// TIA Portal project "智能仓库" (V16)

(* hardware
DEVICE "S7-1200 station_1"  S7-1200 Station
   slot 0: "Rack_0"  S7-1200 Rack  Rack  V1.0
   slot 1: "PLC_1"  CPU 1214C DC/DC/Rly  6ES7 214-1HG40-0XB0  V4.4
DEVICE "HMI_2"  TP700 Comfort
   slot 0: "HMI_2"  TP700 Comfort  6AV2 124-0GC01-0AX0  16.0.0.0
   slot 1: "HMI_RT_2"  TP700 Comfort  6AV2 124-0GC01-0AX0  16.0.0.0
   slot 5: "HMI_2.IE_CP_1"  PROFINET Interface  16.0.0.0
      slot 1: "PROFINET Interface_1"  PROFINET Interface
         slot 1: "Port_1"  Port
         slot 2: "Port_2"  Port
   slot 7: "HMI_2.MPI/DP_CP_1"  MPI/DP Interface  16.0.0.0
*)

// ===== PLC "PLC_1"  CPU 1214C DC/DC/Rly =====

VAR_GLOBAL   // PLC tag table "默认变量表"
   "System_Byte" AT %MB1 : Byte;
   "FirstScan" AT %M1.0 : Bool;
   "DiagStatusUpdate" AT %M1.1 : Bool;
   "AlwaysTRUE" AT %M1.2 : Bool;
   "AlwaysFALSE" AT %M1.3 : Bool;
   "System_Byte(1)" AT %MB1 : Byte;
   "Clock_Byte" AT %MB0 : Byte;
   "Clock_10Hz" AT %M0.0 : Bool;
   "Clock_5Hz" AT %M0.1 : Bool;
   "Clock_2.5Hz" AT %M0.2 : Bool;
   "Clock_2Hz" AT %M0.3 : Bool;
   "Clock_1.25Hz" AT %M0.4 : Bool;
   "Clock_1Hz" AT %M0.5 : Bool;
   "Clock_0.625Hz" AT %M0.6 : Bool;
   "Clock_0.5Hz" AT %M0.7 : Bool;
   "入库手/自动开关" AT %M10.0 : Bool;
   "自动入库读取当前数组的数据" AT %MB30 : Byte;
   "手动入库读取当前数组的数据" AT %MB34 : Byte;
   "动画列表" AT %MW100 : Int;
   "自动运行指示灯" AT %M10.1 : Bool;
   "手动运行指示灯" AT %M10.2 : Bool;
   "手动出库读取当前数组的数据" AT %MB38 : Byte;
   "自动出库读取当前数组的数据" AT %MB42 : Byte;
   "出库/入库切换开关" AT %M10.3 : Bool;
   "入库指示灯" AT %M10.4 : Bool;
   "出库指示灯" AT %M10.5 : Bool;
   "自动/手动出库开关" AT %M10.6 : Bool;
   "手动出库指示灯" AT %M10.7 : Bool;
   "自动出库指示灯" AT %M11.0 : Bool;
   "启动入库" AT %M100.0 : Bool;
   "启动出库" AT %M100.1 : Bool;
END_VAR

VAR_GLOBAL   // PLC tag table "factory  io"
   "伸出收料到位" AT %I2.0 : Bool;
   "叉车在中间" AT %I2.1 : Bool;
   "伸出放料到位" AT %I2.2 : Bool;
   "物料到位检测信号" AT %I2.3 : Bool;
   "检测物料开关" AT %I2.4 : Bool;
   "MovingX" AT %I2.5 : Bool;
   "Moving Z" AT %I2.6 : Bool;
   "启动" AT %I2.7 : Bool;
   "停止" AT %I3.0 : Bool;
   "出料检测传感器" AT %I3.1 : Bool;
   "显示屏传感器" AT %I3.2 : Bool;
   "复位" AT %I3.3 : Bool;
   "急停" AT %I3.4 : Bool;
   "手动模式" AT %I3.5 : Bool;
   "自动模式" AT %I3.6 : Bool;
   "FACTORY I/O (Running)" AT %I4.1 : Bool;
   "一段电机" AT %Q2.0 : Bool;
   "二段电机" AT %Q2.1 : Bool;
   "伸出取料" AT %Q2.2 : Bool;
   "叉车上升" AT %Q2.3 : Bool;
   "发料" AT %Q2.4 : Bool;
   "伸出放料" AT %Q2.5 : Bool;
   "绿色" AT %Q2.6 : Bool;
   "红色" AT %Q2.7 : Bool;
   "三段电机" AT %Q3.0 : Bool;
   "四段电机" AT %Q3.1 : Bool;
   "出料" AT %Q3.2 : Bool;
   "移动目标" AT %QD30 : DInt;
END_VAR

// folder: 数据块

DATA_BLOCK "全局数据块"   // DB1
{ S7_Optimized_Access := 'TRUE' }
VERSION : 0.1
   VAR
      公共数据 : Struct
         物料存储的状态 : Array[1..54] of Byte;
         定时器 : Array[1..10] of IEC_TIMER;
         沿时 : Array[1..10] of Bool;
         中间变量1 : Bool;
      END_STRUCT;
      自动入库 : Struct
         置位复位优先指令 : Array[1..10] of Bool;
         定时器 : Array[1..10] of IEC_TIMER;
         放料数目 : DInt;
         沿时指令 : Array[1..10] of Bool;
         完成标志位 : Bool;
         有料标志位 : Bool;
         无料标志位 : Bool;
      END_STRUCT;
      手动入库 : Struct
         设置取料第几行 : DInt;
         设置取料第几列 : DInt;
         取料第几行 : DInt;
         取料第几列 : DInt;
         取料位置 : DInt;
         空位启动标志位 : Bool;
         手动入库开关 : Bool;
         SR : Array[1..10] of Bool;
         手动定时器 : Array[1..10] of IEC_TIMER;
         沿时指令 : Array[1..10] of Bool;
         手动入库完成标志位 : Bool;
      END_STRUCT;
      动画列表 : Int := 0;
      动画切换 : Struct
         主页 : Bool;
         入库 : Bool;
         出库 : Bool;
         系统设置 : Bool;
         io : Bool;
         注销 : Bool;
         沿 : Array[1..10] of Bool;
      END_STRUCT;
      手动出库 : Struct
         设置取料第几行 : DInt;
         设置取料第几列 : DInt;
         取料第几行 : DInt;
         取料第几列 : DInt;
         取料位置 : DInt;
         空位启动标志位 : Bool;
         手动出库完成标志位 : Bool;
         手动出库完成标志位_1 : Bool;
         手动出库开关 : Bool;
         SR : Array[1..10] of Bool;
         定时器 : Array[1..10] of IEC_TIMER;
         处理双线圈 : Array[1..2] of Bool;
         沿时 : Array[1..10] of Bool;
      END_STRUCT;
      自动出库 : Struct
         出料数目 : DInt;
         置位复位优先指令 : Array[1..10] of Bool;
         定时器 : Array[1..10] of IEC_TIMER;
         沿时指令 : Array[1..10] of Bool;
         完成标志位 : Bool;
         完成标志位_1 : Bool;
         有料标志位 : Bool;
         无料标志位 : Bool;
         双线圈 : Array[0..1] of Bool;
      END_STRUCT;
   END_VAR
BEGIN
   // 自动入库.置位复位优先指令[1] : 1
   // 自动入库.定时器[1] : 1
   // 自动入库.定时器[2] : 1
   // 自动入库.置位复位优先指令[2] : 1
   // 自动入库.定时器[3] : 1
   // 自动入库.置位复位优先指令[3] : 1
   // 自动入库.定时器[4] : 1
   // 自动入库.沿时指令[1] : 1
   // 自动入库.沿时指令[2] : 1
   // 自动入库.定时器[5] : 1
   // 自动入库.定时器[6] : 1
   // 自动入库.置位复位优先指令[4] : 1
   // 自动入库.沿时指令[3] : 1
   // 手动出库.定时器[1] : 1
   // 手动出库.定时器[2] : 1
   // 手动出库.定时器[3] : 1
   // 手动出库.定时器[4] : 1
   // 手动出库.定时器[5] : 1
   // 手动出库.定时器[6] : 1
   // 自动出库.置位复位优先指令[1] : 1
   // 自动出库.置位复位优先指令[2] : 1
   // 自动出库.置位复位优先指令[3] : 1
   // 自动出库.置位复位优先指令[4] : 1
   // 自动出库.定时器[1] : 1
   // 自动出库.定时器[2] : 1
   // 自动出库.定时器[3] : 1
   // 自动出库.定时器[4] : 1
   // 自动出库.定时器[5] : 1
   // 自动出库.定时器[6] : 1
   // 自动出库.沿时指令[1] : 1
   // 自动出库.沿时指令[2] : 1
   // 自动出库.沿时指令[3] : 1
END_DATA_BLOCK

// folder: (top level)

FUNCTION "MHJ-PLC-Lab-Function-S71200" : Void   // FC9000, SCL
{ S7_Optimized_Access := 'TRUE' }
VERSION : 0.1
   VAR_TEMP
      rdTimeReturn : Int;
      outputTime : DTL;
      SyncVal : Byte;
      forVal : Int;
      forVal_2 : Int;
      Value : Byte;
   END_VAR
   VAR CONSTANT
      CompVal : Byte := 16#34;
      Value_01 : Byte := 16#11;
      Value_01_DW : DWord := 16#A165_D992;
      Value_02_DW : DWord := 16#58BE_4401;
   END_VAR
BEGIN

   #Value:=PEEK(area := 16#82,
        dbNumber := 0,
        byteOffset := 511);
   #Value := #Value + 1;

   POKE(area := 16#82,
        dbNumber := 0,
        byteOffset := 511,
        value := #Value);

   POKE(area:=16#81,
        dbNumber:=0,
        byteOffset:=1016,
        value:=#Value_01_DW);
   POKE(area := 16#81,
        dbNumber := 0,
        byteOffset := 1020,
        value := #Value_02_DW);

   POKE(area := 16#81,
        dbNumber := 0,
        byteOffset := 511,
        value := B#16#00);

   FOR #forVal := 0 TO 120 DO
       FOR #forVal_2:=0 TO 10 DO
           #rdTimeReturn:=RD_SYS_T(#outputTime);
           #rdTimeReturn := WR_SYS_T(#outputTime);
           #rdTimeReturn := RD_SYS_T(#outputTime);
           #rdTimeReturn := WR_SYS_T(#outputTime);
       END_FOR;
       #SyncVal:= PEEK(area := 16#81,
                      dbNumber := 0,
                      byteOffset := 511);
       IF #SyncVal = #CompVal THEN
          GOTO M_1;
       END_IF;
   END_FOR;
   RETURN;

   M_1:
   POKE(area := 16#81,
        dbNumber := 0,
        byteOffset := 511,
        value := B#16#0);
END_FUNCTION

ORGANIZATION_BLOCK "Main"   // OB1, LAD, ProgramCycle
TITLE = "Main Program Sweep (Cycle)"
{ S7_Optimized_Access := 'TRUE' }
VERSION : 0.1
   VAR_INPUT
      Initial_Call : Bool;   // Initial call of this OB
      Remanence : Bool;   // =True, if remanent data are available
   END_VAR
   VAR_TEMP   // added for the SCL form of the ladder/FBD networks
      _w1 : Bool;
      _w2 : Bool;
      _w3 : Bool;
      _w4 : Bool;
      _w5 : Bool;
      _w6 : Bool;
      _w7 : Bool;
      _w8 : Bool;
      _w9 : Bool;
   END_VAR
BEGIN

REGION Network 1
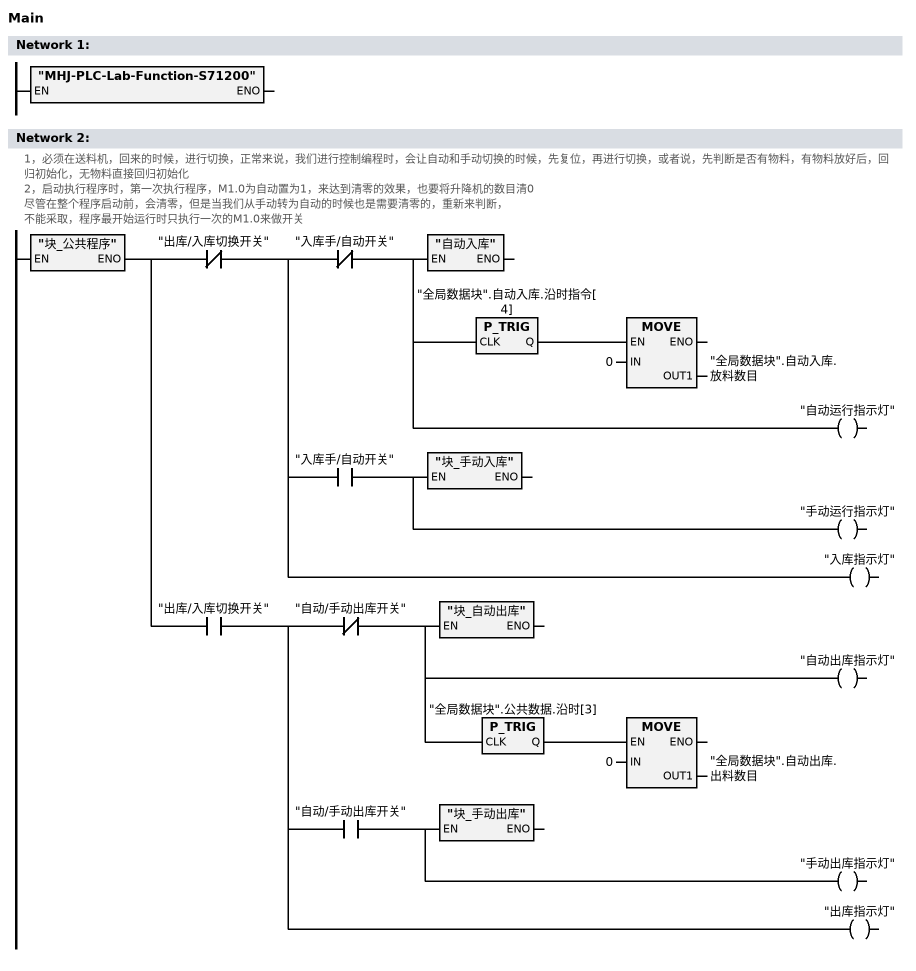
   RUNG wire#powerrail
      "MHJ-PLC-Lab-Function-S71200"()
   END_RUNG
   // the same network as SCL:
   "MHJ-PLC-Lab-Function-S71200"();
END_REGION

REGION Network 2
   // 1，必须在送料机，回来的时候，进行切换，正常来说，我们进行控制编程时，会让自动和手动切换的时候，先复位，再进行切换，或者说，先判断是否有物料，有物料放好后，回归初始化，无物料直接回归初始化
   // 2，启动执行程序时，第一次执行程序，M1.0为自动置为1，来达到清零的效果，也要将升降机的数目清0
   // 尽管在整个程序启动前，会清零，但是当我们从手动转为自动的时候也是需要清零的，重新来判断，
   // 不能采取，程序最开始运行时只执行一次的M1.0来做开关
   RUNG wire#powerrail
      "块_公共程序"()
      wire#w1
      I_Contact( "出库/入库切换开关" )
      wire#w2
      I_Contact( "入库手/自动开关" )
      wire#w3
      "自动入库"()
   END_RUNG
   RUNG wire#w3
      P_Trig( "全局数据块".自动入库.沿时指令[4] )
      Move(in := 0, out1 => "全局数据块".自动入库.放料数目)
   END_RUNG
   RUNG wire#w3
      Coil( "自动运行指示灯" )
   END_RUNG
   RUNG wire#w2
      Contact( "入库手/自动开关" )
      wire#w4
      "块_手动入库"()
   END_RUNG
   RUNG wire#w4
      Coil( "手动运行指示灯" )
   END_RUNG
   RUNG wire#w2
      Coil( "入库指示灯" )
   END_RUNG
   RUNG wire#w1
      Contact( "出库/入库切换开关" )
      wire#w5
      I_Contact( "自动/手动出库开关" )
      wire#w6
      "块_自动出库"()
   END_RUNG
   RUNG wire#w6
      Coil( "自动出库指示灯" )
   END_RUNG
   RUNG wire#w6
      P_Trig( "全局数据块".公共数据.沿时[3] )
      Move(in := 0, out1 => "全局数据块".自动出库.出料数目)
   END_RUNG
   RUNG wire#w5
      Contact( "自动/手动出库开关" )
      wire#w7
      "块_手动出库"()
   END_RUNG
   RUNG wire#w7
      Coil( "手动出库指示灯" )
   END_RUNG
   RUNG wire#w5
      Coil( "出库指示灯" )
   END_RUNG
   // the same network as SCL:
   "块_公共程序"(ENO => #_w1);
   #_w2 := #_w1 AND NOT "出库/入库切换开关";
   #_w3 := #_w2 AND NOT "入库手/自动开关";
   IF #_w3 THEN "自动入库"(); END_IF;
   #_w4 := #_w3 AND NOT "全局数据块".自动入库.沿时指令[4];   // rising edge
   "全局数据块".自动入库.沿时指令[4] := #_w3;
   IF #_w4 THEN "全局数据块".自动入库.放料数目 := 0; END_IF;
   "自动运行指示灯" := #_w3;
   #_w5 := #_w2 AND "入库手/自动开关";
   IF #_w5 THEN "块_手动入库"(); END_IF;
   "手动运行指示灯" := #_w5;
   "入库指示灯" := #_w2;
   #_w6 := #_w1 AND "出库/入库切换开关";
   #_w7 := #_w6 AND NOT "自动/手动出库开关";
   IF #_w7 THEN "块_自动出库"(); END_IF;
   "自动出库指示灯" := #_w7;
   #_w8 := #_w7 AND NOT "全局数据块".公共数据.沿时[3];   // rising edge
   "全局数据块".公共数据.沿时[3] := #_w7;
   IF #_w8 THEN "全局数据块".自动出库.出料数目 := 0; END_IF;
   #_w9 := #_w6 AND "自动/手动出库开关";
   IF #_w9 THEN "块_手动出库"(); END_IF;
   "手动出库指示灯" := #_w9;
   "出库指示灯" := #_w6;
END_REGION
END_ORGANIZATION_BLOCK

// folder: 公共程序

FUNCTION "块_公共程序" : Void   // FC3, LAD
{ S7_Optimized_Access := 'TRUE' }
VERSION : 0.1
   VAR_TEMP   // added for the SCL form of the ladder/FBD networks
      _w1 : Bool;
      _w2 : Bool;
      _w3 : Bool;
      _w4 : Bool;
      _w5 : Bool;
   END_VAR
BEGIN

REGION Network 1: 初始化
   // 启动执行程序时，第一次执行程序，M1.0为自动置为1，来达到清零的效果，也要将升降机的数目清0
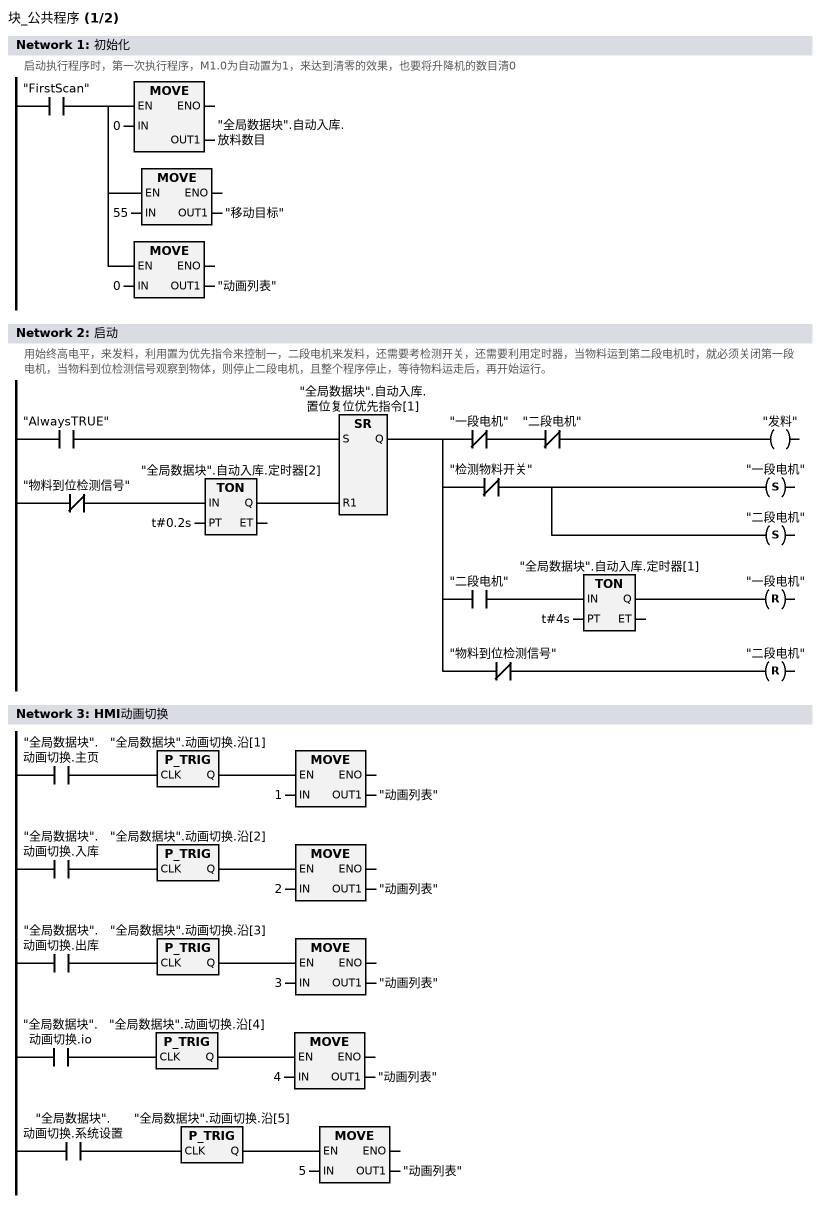
   RUNG wire#powerrail
      Contact( "FirstScan" )
      wire#w1
      Move(in := 0, out1 => "全局数据块".自动入库.放料数目)
   END_RUNG
   RUNG wire#w1
      Move(in := 55, out1 => "移动目标")
   END_RUNG
   RUNG wire#w1
      Move(in := 0, out1 => "动画列表")
   END_RUNG
   // the same network as SCL:
   IF "FirstScan" THEN
       "全局数据块".自动入库.放料数目 := 0;
       "移动目标" := 55;
       "动画列表" := 0;
   END_IF;
END_REGION

REGION Network 2: 启动
   // 用始终高电平，来发料，利用置为优先指令来控制一，二段电机来发料，还需要考检测开关，还需要利用定时器，当物料运到第二段电机时，就必须关闭第一段电机，当物料到位检测信号观察到物体，则停止二段电机，且整个程序停止，等待物料运走后，再开始运行。
   "全局数据块".自动入库.定时器[2].TON(IN := NOT "物料到位检测信号", PT := t#0.2s);
   IF "AlwaysTRUE" THEN
       "全局数据块".自动入库.置位复位优先指令[1] := TRUE;   // SR flip-flop
   END_IF;
   IF "全局数据块".自动入库.定时器[2].Q THEN "全局数据块".自动入库.置位复位优先指令[1] := FALSE; END_IF;
   "发料" := "全局数据块".自动入库.置位复位优先指令[1] AND NOT "一段电机" AND NOT "二段电机";
   IF "全局数据块".自动入库.置位复位优先指令[1] AND NOT "检测物料开关" THEN
       "一段电机" := TRUE;
       "二段电机" := TRUE;
   END_IF;
   "全局数据块".自动入库.定时器[1].TON(IN := "全局数据块".自动入库.置位复位优先指令[1] AND "二段电机", PT := t#4s);
   IF "全局数据块".自动入库.定时器[1].Q THEN "一段电机" := FALSE; END_IF;
   IF "全局数据块".自动入库.置位复位优先指令[1] AND NOT "物料到位检测信号" THEN "二段电机" := FALSE; END_IF;
END_REGION

REGION Network 3: HMI动画切换
   RUNG wire#powerrail
      Contact( "全局数据块".动画切换.主页 )
      P_Trig( "全局数据块".动画切换.沿[1] )
      Move(in := 1, out1 => "动画列表")
   END_RUNG
   RUNG wire#powerrail
      Contact( "全局数据块".动画切换.入库 )
      P_Trig( "全局数据块".动画切换.沿[2] )
      Move(in := 2, out1 => "动画列表")
   END_RUNG
   RUNG wire#powerrail
      Contact( "全局数据块".动画切换.出库 )
      P_Trig( "全局数据块".动画切换.沿[3] )
      Move(in := 3, out1 => "动画列表")
   END_RUNG
   RUNG wire#powerrail
      Contact( "全局数据块".动画切换.io )
      P_Trig( "全局数据块".动画切换.沿[4] )
      Move(in := 4, out1 => "动画列表")
   END_RUNG
   RUNG wire#powerrail
      Contact( "全局数据块".动画切换.系统设置 )
      P_Trig( "全局数据块".动画切换.沿[5] )
      Move(in := 5, out1 => "动画列表")
   END_RUNG
   // the same network as SCL:
   #_w1 := "全局数据块".动画切换.主页 AND NOT "全局数据块".动画切换.沿[1];   // rising edge
   "全局数据块".动画切换.沿[1] := "全局数据块".动画切换.主页;
   IF #_w1 THEN "动画列表" := 1; END_IF;
   #_w2 := "全局数据块".动画切换.入库 AND NOT "全局数据块".动画切换.沿[2];   // rising edge
   "全局数据块".动画切换.沿[2] := "全局数据块".动画切换.入库;
   IF #_w2 THEN "动画列表" := 2; END_IF;
   #_w3 := "全局数据块".动画切换.出库 AND NOT "全局数据块".动画切换.沿[3];   // rising edge
   "全局数据块".动画切换.沿[3] := "全局数据块".动画切换.出库;
   IF #_w3 THEN "动画列表" := 3; END_IF;
   #_w4 := "全局数据块".动画切换.io AND NOT "全局数据块".动画切换.沿[4];   // rising edge
   "全局数据块".动画切换.沿[4] := "全局数据块".动画切换.io;
   IF #_w4 THEN "动画列表" := 4; END_IF;
   #_w5 := "全局数据块".动画切换.系统设置 AND NOT "全局数据块".动画切换.沿[5];   // rising edge
   "全局数据块".动画切换.沿[5] := "全局数据块".动画切换.系统设置;
   IF #_w5 THEN "动画列表" := 5; END_IF;
END_REGION

REGION Network 4: 出料
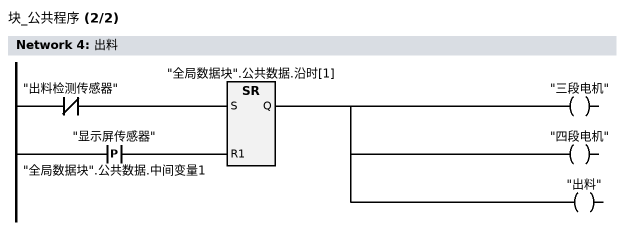
   RUNG wire#powerrail
      I_Contact( "出料检测传感器" )
      S_SR(operand := "全局数据块".公共数据.沿时[1], r1 := wire#w1)
      wire#w2
      Coil( "三段电机" )
   END_RUNG
   RUNG wire#powerrail
      P_Contact(operand := "显示屏传感器", bit := "全局数据块".公共数据.中间变量1)
   END_RUNG wire#w1
   RUNG wire#w2
      Coil( "四段电机" )
   END_RUNG
   RUNG wire#w2
      Coil( "出料" )
   END_RUNG
   // the same network as SCL:
   #_w1 := "显示屏传感器" AND NOT "全局数据块".公共数据.中间变量1;   // rising edge of "显示屏传感器"
   "全局数据块".公共数据.中间变量1 := "显示屏传感器";
   IF NOT "出料检测传感器" THEN
       "全局数据块".公共数据.沿时[1] := TRUE;   // SR flip-flop
   END_IF;
   IF #_w1 THEN "全局数据块".公共数据.沿时[1] := FALSE; END_IF;
   "三段电机" := "全局数据块".公共数据.沿时[1];
   "四段电机" := "全局数据块".公共数据.沿时[1];
   "出料" := "全局数据块".公共数据.沿时[1];
END_REGION
END_FUNCTION

// folder: 复位

FUNCTION "块_复位" : Void   // FC6, LAD
{ S7_Optimized_Access := 'TRUE' }
VERSION : 0.1
BEGIN
END_FUNCTION

// folder: 手动入库

FUNCTION "块_手动入库" : Void   // FC1, LAD
{ S7_Optimized_Access := 'TRUE' }
VERSION : 0.1
   VAR_TEMP   // added for the SCL form of the ladder/FBD networks
      _w1 : Bool;
      _w2 : Bool;
      _w3 : Bool;
   END_VAR
BEGIN

REGION Network 1: 设置放料的地址
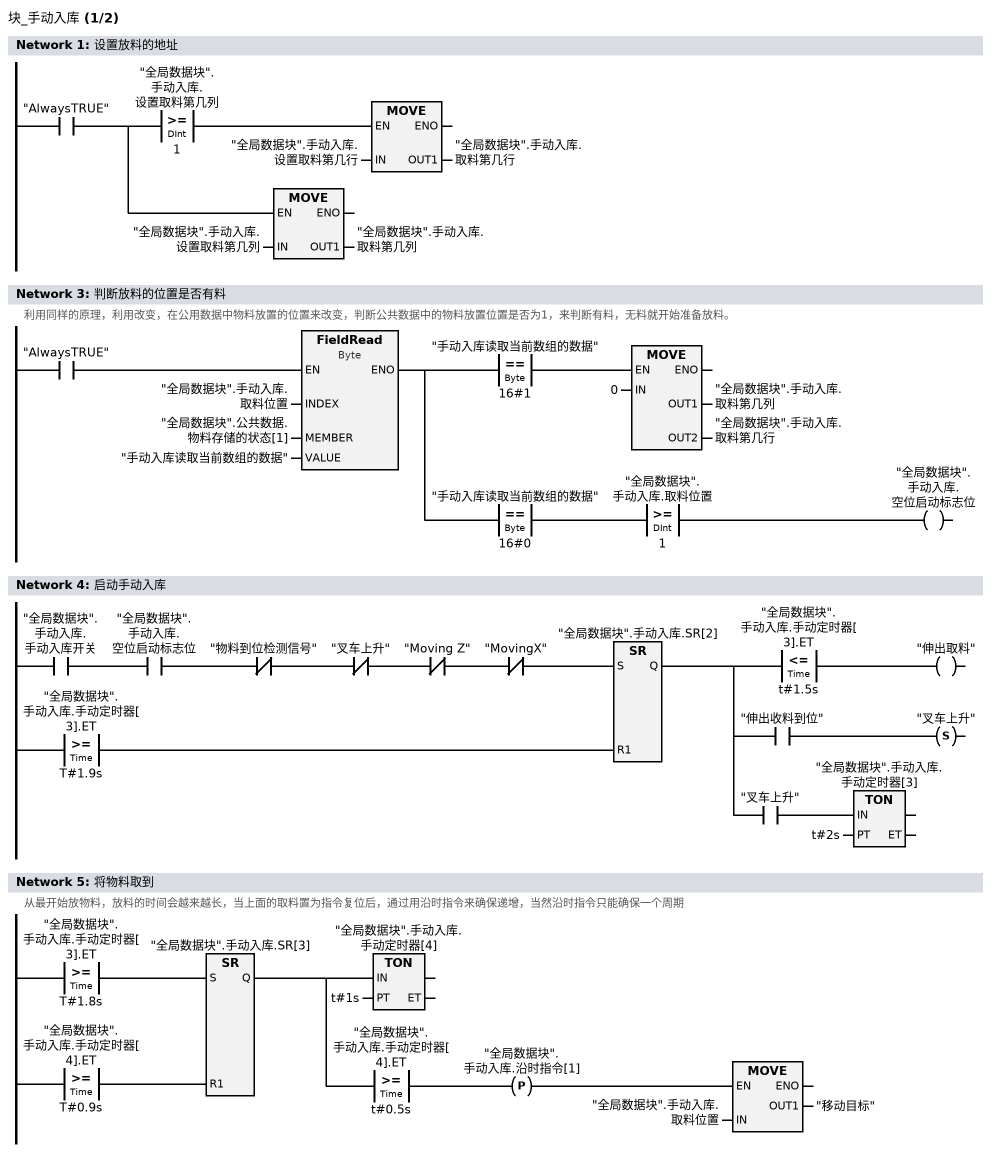
   RUNG wire#powerrail
      Contact( "AlwaysTRUE" )
      wire#w1
      { S7_Templates := "SrcType := DInt" } GE_Contact(in1 := "全局数据块".手动入库.设置取料第几列, in2 := 1)
      Move(in := "全局数据块".手动入库.设置取料第几行, out1 => "全局数据块".手动入库.取料第几行)
   END_RUNG
   RUNG wire#w1
      Move(in := "全局数据块".手动入库.设置取料第几列, out1 => "全局数据块".手动入库.取料第几列)
   END_RUNG
   // the same network as SCL:
   IF "AlwaysTRUE" AND ("全局数据块".手动入库.设置取料第几列 >= 1) THEN "全局数据块".手动入库.取料第几行 := "全局数据块".手动入库.设置取料第几行; END_IF;
   IF "AlwaysTRUE" THEN "全局数据块".手动入库.取料第几列 := "全局数据块".手动入库.设置取料第几列; END_IF;
END_REGION

REGION Network 2 (SCL): 这里利用的SCL语言用来计算，
   // 其实可以用，我认为用综合计算指令也可以得到这样的结果将列设置为x，将行设置y
   // 通过（x-1）9+y就可以得到具体位置
   //相当于c语言编程一样
   //将结果放在前面，计算的公式放在后面
   //程序的格式，必须用英文大写
   //还需要写一个判断语句
   //IF "全局数据块".手动入库.取料第几行 = 0 AND "全局数据块".手动入库.取料第几列 = 0 OR "全局数据块".手动入库.取料位置 > 54 THEN
   // "全局数据块".手动入库.取料位置 := 0;
   //END_IF;
   //IF  "全局数据块".手动入库.取料第几行 > 0 AND "全局数据块".手动入库.取料第几列 > 0AND"全局数据块".手动入库.取料第几行 <7 AND "全局数据块".手动入库.取料第几列 <10 THEN
       //"全局数据块".手动入库.取料位置 := ("全局数据块".手动入库.取料第几行 - 1) * 9 +"全局数据块".手动入库.取料第几列 ;
   //END_IF;
   IF  "全局数据块".手动入库.取料第几行 = 0 AND "全局数据块".手动入库.取料第几列 = 0 OR "全局数据块".手动入库.取料位置 > 54  THEN
       "全局数据块".手动入库.取料位置 := 0;
       "全局数据块".手动入库.设置取料第几行 := 0;
       "全局数据块".手动入库.设置取料第几列 := 0;
   ELSE
       "全局数据块".手动入库.取料位置 := ("全局数据块".手动入库.取料第几行 - 1) * 9 + "全局数据块".手动入库.取料第几列;
   END_IF;
END_REGION

REGION Network 3: 判断放料的位置是否有料
   // 利用同样的原理，利用改变，在公用数据中物料放置的位置来改变，判断公共数据中的物料放置位置是否为1，来判断有料，无料就开始准备放料。
   // no SCL statement known for FieldRead: written as a call
   // ENO of a box is taken as its EN; it also drops when the box reports an error
   #_w1 := "AlwaysTRUE";
   IF #_w1 THEN
       FieldRead(index := "全局数据块".手动入库.取料位置, member := "全局数据块".公共数据.物料存储的状态[1], value := "手动入库读取当前数组的数据");
   END_IF;
   IF #_w1 AND ("手动入库读取当前数组的数据" = 16#1) THEN
       "全局数据块".手动入库.取料第几列 := 0;
       "全局数据块".手动入库.取料第几行 := 0;
   END_IF;
   "全局数据块".手动入库.空位启动标志位 := #_w1 AND ("手动入库读取当前数组的数据" = 16#0) AND ("全局数据块".手动入库.取料位置 >= 1);
END_REGION

REGION Network 4: 启动手动入库
   IF "全局数据块".手动入库.手动入库开关 AND "全局数据块".手动入库.空位启动标志位 AND NOT "物料到位检测信号" AND NOT "叉车上升" AND NOT "Moving Z" AND NOT "MovingX" THEN
       "全局数据块".手动入库.SR[2] := TRUE;   // SR flip-flop
   END_IF;
   IF "全局数据块".手动入库.手动定时器[3].ET >= T#1.9s THEN "全局数据块".手动入库.SR[2] := FALSE; END_IF;
   "伸出取料" := "全局数据块".手动入库.SR[2] AND ("全局数据块".手动入库.手动定时器[3].ET <= t#1.5s);
   IF "全局数据块".手动入库.SR[2] AND "伸出收料到位" THEN "叉车上升" := TRUE; END_IF;
   "全局数据块".手动入库.手动定时器[3].TON(IN := "全局数据块".手动入库.SR[2] AND "叉车上升", PT := t#2s);
END_REGION

REGION Network 5: 将物料取到
   // 从最开始放物料，放料的时间会越来越长，当上面的取料置为指令复位后，通过用沿时指令来确保递增，当然沿时指令只能确保一个周期
   IF "全局数据块".手动入库.手动定时器[3].ET >= T#1.8s THEN
       "全局数据块".手动入库.SR[3] := TRUE;   // SR flip-flop
   END_IF;
   IF "全局数据块".手动入库.手动定时器[4].ET >= T#0.9s THEN "全局数据块".手动入库.SR[3] := FALSE; END_IF;
   "全局数据块".手动入库.手动定时器[4].TON(IN := "全局数据块".手动入库.SR[3], PT := t#1s);
   #_w1 := "全局数据块".手动入库.SR[3] AND ("全局数据块".手动入库.手动定时器[4].ET >= t#0.5s);
   #_w2 := #_w1 AND NOT "全局数据块".手动入库.沿时指令[1];   // rising edge
   "全局数据块".手动入库.沿时指令[1] := #_w1;
   IF #_w2 THEN "移动目标" := "全局数据块".手动入库.取料位置; END_IF;
END_REGION

REGION Network 6: 入库
   // 需要在这里对于外面放入的物料进行记录.我想的是通过写入域，再加上下标的增加，就可以达到记录的目的,但是需要将两边的数据类型变为一致的，需要进行一个转换指令。老师讲的是通过move指令，可以改变写入，地址那个变换的值，当然最小的存储单位是byte，我所用的是byte所以，我无法进行将大的改变为小的，来达到每一个记录
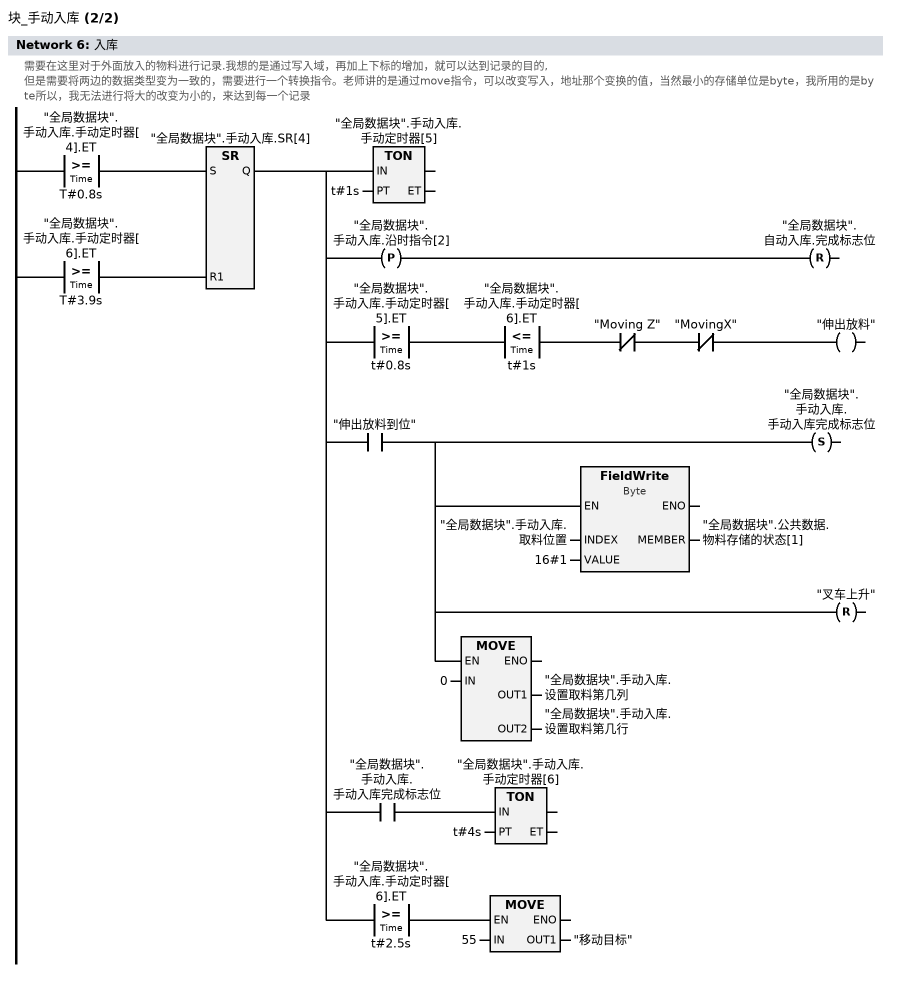
   // no SCL statement known for FieldWrite: written as a call
   IF "全局数据块".手动入库.手动定时器[4].ET >= T#0.8s THEN
       "全局数据块".手动入库.SR[4] := TRUE;   // SR flip-flop
   END_IF;
   IF "全局数据块".手动入库.手动定时器[6].ET >= T#3.9s THEN "全局数据块".手动入库.SR[4] := FALSE; END_IF;
   "全局数据块".手动入库.手动定时器[5].TON(IN := "全局数据块".手动入库.SR[4], PT := t#1s);
   #_w1 := "全局数据块".手动入库.SR[4] AND NOT "全局数据块".手动入库.沿时指令[2];   // rising edge
   "全局数据块".手动入库.沿时指令[2] := "全局数据块".手动入库.SR[4];
   IF #_w1 THEN "全局数据块".自动入库.完成标志位 := FALSE; END_IF;
   "伸出放料" := "全局数据块".手动入库.SR[4] AND ("全局数据块".手动入库.手动定时器[5].ET >= t#0.8s) AND ("全局数据块".手动入库.手动定时器[6].ET <= t#1s) AND NOT "Moving Z" AND NOT "MovingX";
   IF "全局数据块".手动入库.SR[4] AND "伸出放料到位" THEN "全局数据块".手动入库.手动入库完成标志位 := TRUE; END_IF;
   #_w2 := "全局数据块".手动入库.SR[4];
   #_w3 := "全局数据块".手动入库.SR[4] AND "伸出放料到位";
   IF #_w3 THEN
       FieldWrite(index := "全局数据块".手动入库.取料位置, value := 16#1, member => "全局数据块".公共数据.物料存储的状态[1]);
       "叉车上升" := FALSE;
       "全局数据块".手动入库.设置取料第几列 := 0;
       "全局数据块".手动入库.设置取料第几行 := 0;
   END_IF;
   "全局数据块".手动入库.手动定时器[6].TON(IN := #_w2 AND "全局数据块".手动入库.手动入库完成标志位, PT := t#4s);
   IF #_w2 AND ("全局数据块".手动入库.手动定时器[6].ET >= t#2.5s) THEN "移动目标" := 55; END_IF;
END_REGION
END_FUNCTION

// folder: 手动出库

FUNCTION "块_手动出库" : Void   // FC4, LAD
{ S7_Optimized_Access := 'TRUE' }
VERSION : 0.1
   VAR_TEMP   // added for the SCL form of the ladder/FBD networks
      _w1 : Bool;
      _w2 : Bool;
   END_VAR
BEGIN

REGION Network 1: 设置放料的地址
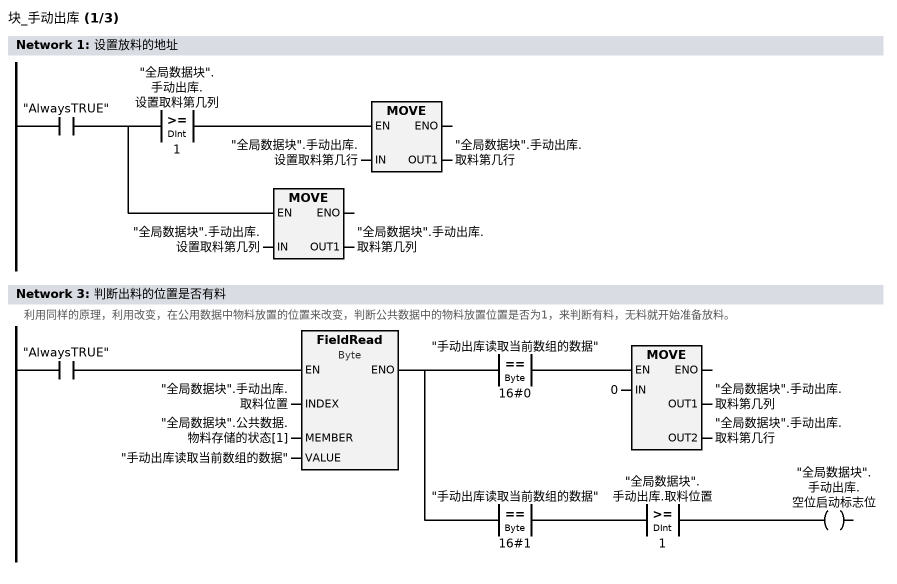
   RUNG wire#powerrail
      Contact( "AlwaysTRUE" )
      wire#w1
      { S7_Templates := "SrcType := DInt" } GE_Contact(in1 := "全局数据块".手动出库.设置取料第几列, in2 := 1)
      Move(in := "全局数据块".手动出库.设置取料第几行, out1 => "全局数据块".手动出库.取料第几行)
   END_RUNG
   RUNG wire#w1
      Move(in := "全局数据块".手动出库.设置取料第几列, out1 => "全局数据块".手动出库.取料第几列)
   END_RUNG
   // the same network as SCL:
   IF "AlwaysTRUE" AND ("全局数据块".手动出库.设置取料第几列 >= 1) THEN "全局数据块".手动出库.取料第几行 := "全局数据块".手动出库.设置取料第几行; END_IF;
   IF "AlwaysTRUE" THEN "全局数据块".手动出库.取料第几列 := "全局数据块".手动出库.设置取料第几列; END_IF;
END_REGION

REGION Network 2 (SCL)
   IF "全局数据块".手动出库.取料第几行 = 0 AND "全局数据块".手动出库.取料第几列 = 0 OR "全局数据块".手动出库.取料位置 > 54 THEN
       "全局数据块".手动出库.取料位置 := 0;
       "全局数据块".手动出库.设置取料第几行 := 0;
       "全局数据块".手动出库.设置取料第几列 := 0;
   ELSE
       "全局数据块".手动出库.取料位置 := ("全局数据块".手动出库.取料第几行 - 1) * 9 + "全局数据块".手动出库.取料第几列;
   END_IF;
END_REGION

REGION Network 3: 判断出料的位置是否有料
   // 利用同样的原理，利用改变，在公用数据中物料放置的位置来改变，判断公共数据中的物料放置位置是否为1，来判断有料，无料就开始准备放料。
   // no SCL statement known for FieldRead: written as a call
   // ENO of a box is taken as its EN; it also drops when the box reports an error
   #_w1 := "AlwaysTRUE";
   IF #_w1 THEN
       FieldRead(index := "全局数据块".手动出库.取料位置, member := "全局数据块".公共数据.物料存储的状态[1], value := "手动出库读取当前数组的数据");
   END_IF;
   IF #_w1 AND ("手动出库读取当前数组的数据" = 16#0) THEN
       "全局数据块".手动出库.取料第几列 := 0;
       "全局数据块".手动出库.取料第几行 := 0;
   END_IF;
   "全局数据块".手动出库.空位启动标志位 := #_w1 AND ("手动出库读取当前数组的数据" = 16#1) AND ("全局数据块".手动出库.取料位置 >= 1);
END_REGION

REGION Network 4: 启动出库
   // 当程序导通，但是动作没有执行 说明双线圈，一般我西环采取 置位复位写程序
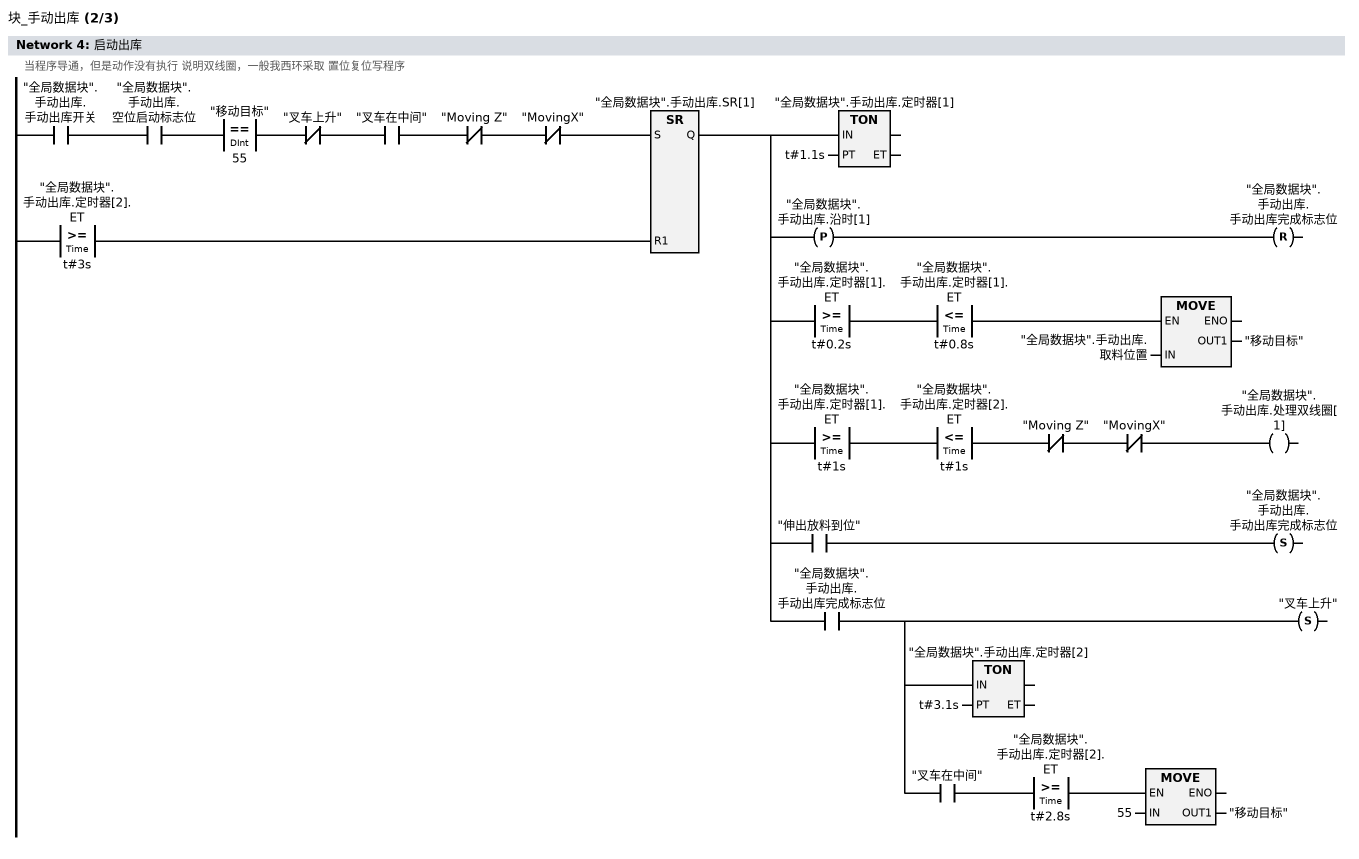
   IF "全局数据块".手动出库.手动出库开关 AND "全局数据块".手动出库.空位启动标志位 AND ("移动目标" = 55) AND NOT "叉车上升" AND "叉车在中间" AND NOT "Moving Z" AND NOT "MovingX" THEN
       "全局数据块".手动出库.SR[1] := TRUE;   // SR flip-flop
   END_IF;
   IF "全局数据块".手动出库.定时器[2].ET >= t#3s THEN "全局数据块".手动出库.SR[1] := FALSE; END_IF;
   "全局数据块".手动出库.定时器[1].TON(IN := "全局数据块".手动出库.SR[1], PT := t#1.1s);
   #_w1 := "全局数据块".手动出库.SR[1] AND NOT "全局数据块".手动出库.沿时[1];   // rising edge
   "全局数据块".手动出库.沿时[1] := "全局数据块".手动出库.SR[1];
   IF #_w1 THEN "全局数据块".手动出库.手动出库完成标志位 := FALSE; END_IF;
   IF "全局数据块".手动出库.SR[1] AND ("全局数据块".手动出库.定时器[1].ET >= t#0.2s) AND ("全局数据块".手动出库.定时器[1].ET <= t#0.8s) THEN
       "移动目标" := "全局数据块".手动出库.取料位置;
   END_IF;
   "全局数据块".手动出库.处理双线圈[1] := "全局数据块".手动出库.SR[1] AND ("全局数据块".手动出库.定时器[1].ET >= t#1s) AND ("全局数据块".手动出库.定时器[2].ET <= t#1s) AND NOT "Moving Z" AND NOT "MovingX";
   IF "全局数据块".手动出库.SR[1] AND "伸出放料到位" THEN "全局数据块".手动出库.手动出库完成标志位 := TRUE; END_IF;
   #_w2 := "全局数据块".手动出库.SR[1] AND "全局数据块".手动出库.手动出库完成标志位;
   IF #_w2 THEN "叉车上升" := TRUE; END_IF;
   "全局数据块".手动出库.定时器[2].TON(IN := #_w2, PT := t#3.1s);
   IF #_w2 AND "叉车在中间" AND ("全局数据块".手动出库.定时器[2].ET >= t#2.8s) THEN "移动目标" := 55; END_IF;
END_REGION

REGION Network 5: 出料
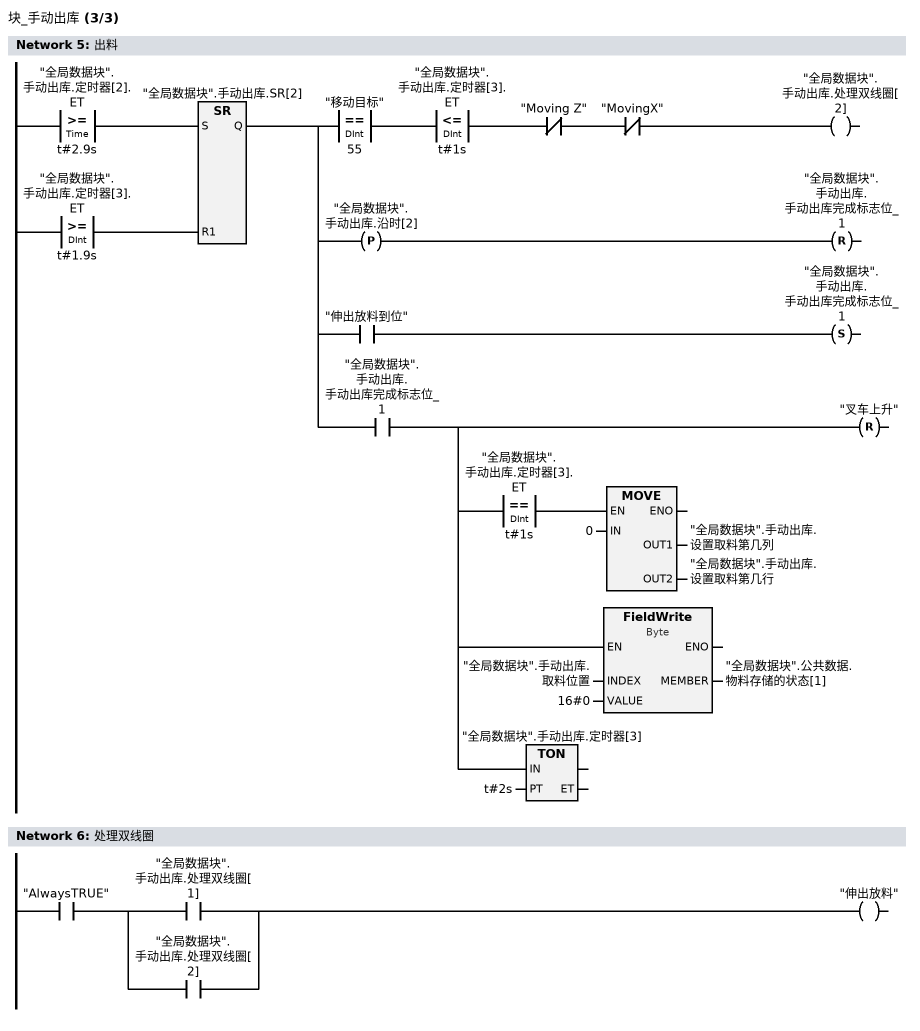
   // no SCL statement known for FieldWrite: written as a call
   IF "全局数据块".手动出库.定时器[2].ET >= t#2.9s THEN
       "全局数据块".手动出库.SR[2] := TRUE;   // SR flip-flop
   END_IF;
   IF "全局数据块".手动出库.定时器[3].ET >= t#1.9s THEN "全局数据块".手动出库.SR[2] := FALSE; END_IF;
   "全局数据块".手动出库.处理双线圈[2] := "全局数据块".手动出库.SR[2] AND ("移动目标" = 55) AND ("全局数据块".手动出库.定时器[3].ET <= t#1s) AND NOT "Moving Z" AND NOT "MovingX";
   #_w1 := "全局数据块".手动出库.SR[2] AND NOT "全局数据块".手动出库.沿时[2];   // rising edge
   "全局数据块".手动出库.沿时[2] := "全局数据块".手动出库.SR[2];
   IF #_w1 THEN "全局数据块".手动出库.手动出库完成标志位_1 := FALSE; END_IF;
   IF "全局数据块".手动出库.SR[2] AND "伸出放料到位" THEN "全局数据块".手动出库.手动出库完成标志位_1 := TRUE; END_IF;
   #_w2 := "全局数据块".手动出库.SR[2] AND "全局数据块".手动出库.手动出库完成标志位_1;
   IF #_w2 THEN "叉车上升" := FALSE; END_IF;
   IF #_w2 AND ("全局数据块".手动出库.定时器[3].ET = t#1s) THEN
       "全局数据块".手动出库.设置取料第几列 := 0;
       "全局数据块".手动出库.设置取料第几行 := 0;
   END_IF;
   IF #_w2 THEN
       FieldWrite(index := "全局数据块".手动出库.取料位置, value := 16#0, member => "全局数据块".公共数据.物料存储的状态[1]);
   END_IF;
   "全局数据块".手动出库.定时器[3].TON(IN := #_w2, PT := t#2s);
END_REGION

REGION Network 6: 处理双线圈
   RUNG wire#powerrail
      Contact( "AlwaysTRUE" )
      wire#w1
      Contact( "全局数据块".手动出库.处理双线圈[1] )
      wire#w2
      Coil( "伸出放料" )
   END_RUNG
   RUNG wire#w1
      Contact( "全局数据块".手动出库.处理双线圈[2] )
   END_RUNG wire#w2
   // the same network as SCL:
   "伸出放料" := "AlwaysTRUE" AND ("全局数据块".手动出库.处理双线圈[1] OR "全局数据块".手动出库.处理双线圈[2]);
END_REGION
END_FUNCTION

// folder: 自动入库

FUNCTION "自动入库" : Void   // FC2, LAD
{ S7_Optimized_Access := 'TRUE' }
VERSION : 0.1
   VAR_TEMP   // added for the SCL form of the ladder/FBD networks
      _w1 : Bool;
      _w2 : Bool;
      _w3 : Bool;
      _w4 : Bool;
      _w5 : Bool;
      _w6 : Bool;
   END_VAR
BEGIN

REGION Network 1: 初始化,
   // 启动执行程序时，第一次执行程序，M1.0为自动置为1，来达到清零的效果，也要将升降机的数目清0
   // 尽管在整个程序启动前，会清零，但是当我们从手动转为自动的时候也是需要清零的，重新来判断，
   // 不能采取，程序最开始运行时只执行一次的M1.0来做开关
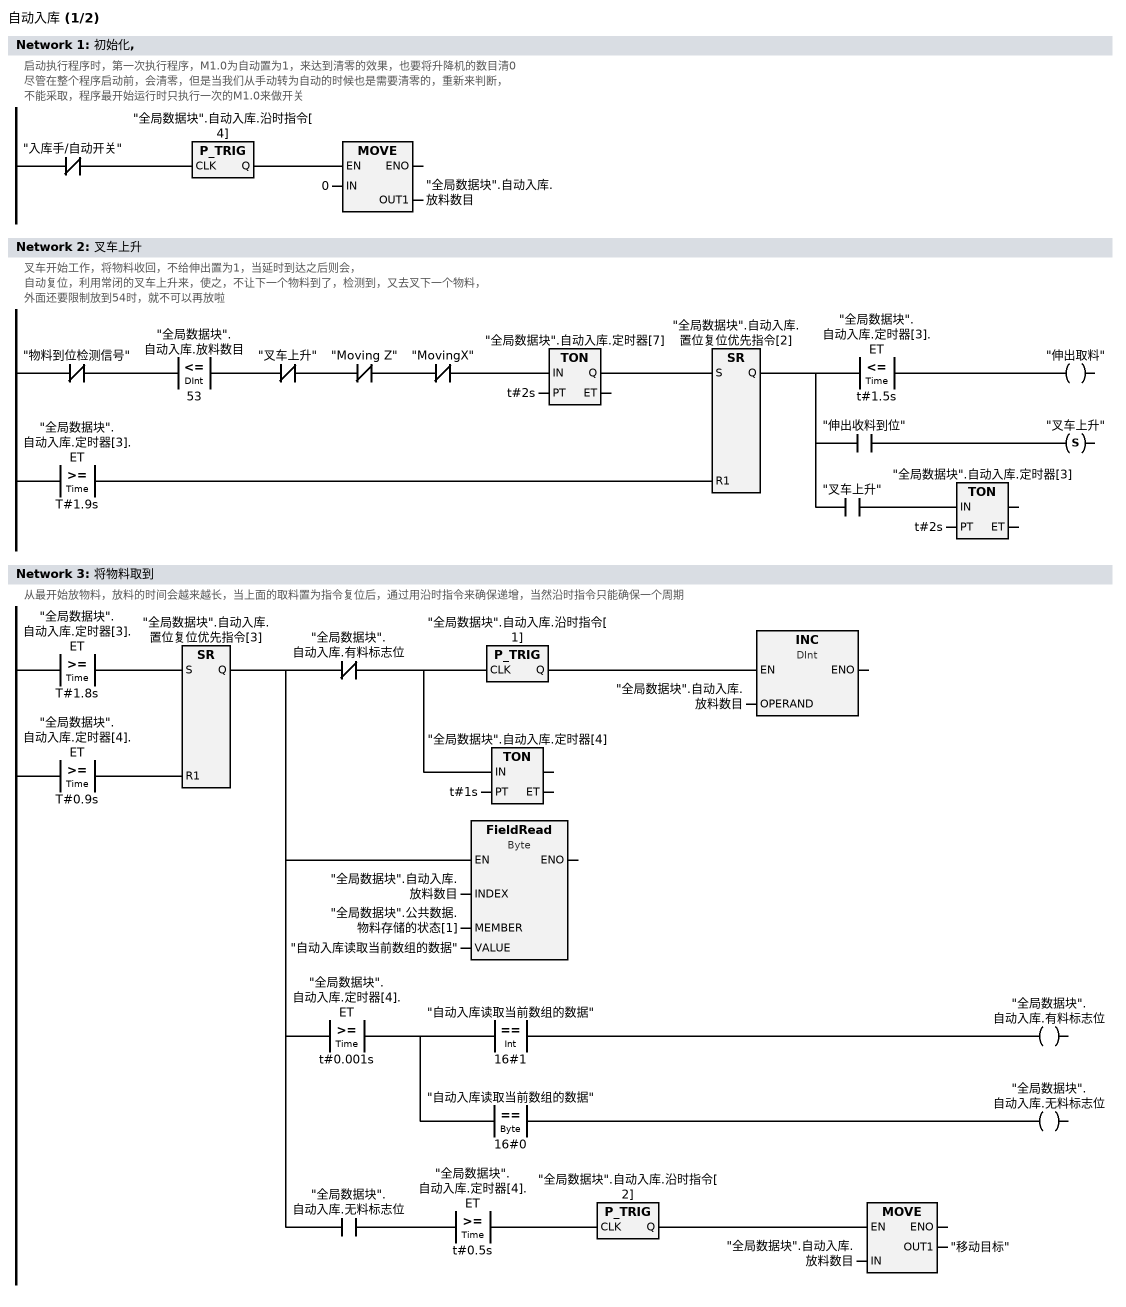
   RUNG wire#powerrail
      I_Contact( "入库手/自动开关" )
      P_Trig( "全局数据块".自动入库.沿时指令[4] )
      Move(in := 0, out1 => "全局数据块".自动入库.放料数目)
   END_RUNG
   // the same network as SCL:
   #_w1 := NOT "入库手/自动开关" AND NOT "全局数据块".自动入库.沿时指令[4];   // rising edge
   "全局数据块".自动入库.沿时指令[4] := NOT "入库手/自动开关";
   IF #_w1 THEN "全局数据块".自动入库.放料数目 := 0; END_IF;
END_REGION

REGION Network 2: 叉车上升
   // 叉车开始工作，将物料收回，不给伸出置为1，当延时到达之后则会，
   // 自动复位，利用常闭的叉车上升来，使之，不让下一个物料到了，检测到，又去叉下一个物料，
   // 外面还要限制放到54时，就不可以再放啦
   "全局数据块".自动入库.定时器[7].TON(IN := NOT "物料到位检测信号" AND ("全局数据块".自动入库.放料数目 <= 53) AND NOT "叉车上升" AND NOT "Moving Z" AND NOT "MovingX",
                           PT := t#2s);
   IF "全局数据块".自动入库.定时器[7].Q THEN
       "全局数据块".自动入库.置位复位优先指令[2] := TRUE;   // SR flip-flop
   END_IF;
   IF "全局数据块".自动入库.定时器[3].ET >= T#1.9s THEN "全局数据块".自动入库.置位复位优先指令[2] := FALSE; END_IF;
   "伸出取料" := "全局数据块".自动入库.置位复位优先指令[2] AND ("全局数据块".自动入库.定时器[3].ET <= t#1.5s);
   IF "全局数据块".自动入库.置位复位优先指令[2] AND "伸出收料到位" THEN "叉车上升" := TRUE; END_IF;
   "全局数据块".自动入库.定时器[3].TON(IN := "全局数据块".自动入库.置位复位优先指令[2] AND "叉车上升", PT := t#2s);
END_REGION

REGION Network 3: 将物料取到
   // 从最开始放物料，放料的时间会越来越长，当上面的取料置为指令复位后，通过用沿时指令来确保递增，当然沿时指令只能确保一个周期
   // no SCL statement known for FieldRead: written as a call
   IF "全局数据块".自动入库.定时器[3].ET >= T#1.8s THEN
       "全局数据块".自动入库.置位复位优先指令[3] := TRUE;   // SR flip-flop
   END_IF;
   IF "全局数据块".自动入库.定时器[4].ET >= T#0.9s THEN "全局数据块".自动入库.置位复位优先指令[3] := FALSE; END_IF;
   #_w1 := "全局数据块".自动入库.置位复位优先指令[3] AND NOT "全局数据块".自动入库.有料标志位;
   #_w2 := #_w1 AND NOT "全局数据块".自动入库.沿时指令[1];   // rising edge
   "全局数据块".自动入库.沿时指令[1] := #_w1;
   IF #_w2 THEN "全局数据块".自动入库.放料数目 := "全局数据块".自动入库.放料数目 + 1; END_IF;
   "全局数据块".自动入库.定时器[4].TON(IN := #_w1, PT := t#1s);
   #_w3 := "全局数据块".自动入库.置位复位优先指令[3];
   IF #_w3 THEN
       FieldRead(index := "全局数据块".自动入库.放料数目, member := "全局数据块".公共数据.物料存储的状态[1], value := "自动入库读取当前数组的数据");
   END_IF;
   #_w4 := #_w3 AND ("全局数据块".自动入库.定时器[4].ET >= t#0.001s);
   "全局数据块".自动入库.有料标志位 := #_w4 AND ("自动入库读取当前数组的数据" = 16#1);
   "全局数据块".自动入库.无料标志位 := #_w4 AND ("自动入库读取当前数组的数据" = 16#0);
   #_w5 := #_w3 AND "全局数据块".自动入库.无料标志位 AND ("全局数据块".自动入库.定时器[4].ET >= t#0.5s);
   #_w6 := #_w5 AND NOT "全局数据块".自动入库.沿时指令[2];   // rising edge
   "全局数据块".自动入库.沿时指令[2] := #_w5;
   IF #_w6 THEN "移动目标" := "全局数据块".自动入库.放料数目; END_IF;
END_REGION

REGION Network 4: 入库
   // 需要在这里对于外面放入的物料进行记录.我想的是通过写入域，再加上下标的增加，就可以达到记录的目的,但是需要将两边的数据类型变为一致的，需要进行一个转换指令。老师讲的是通过move指令，可以改变写入，地址那个变换的值，当然最小的存储单位是byte，我所用的是byte所以，我无法进行将大的改变为小的，来达到每一个记录
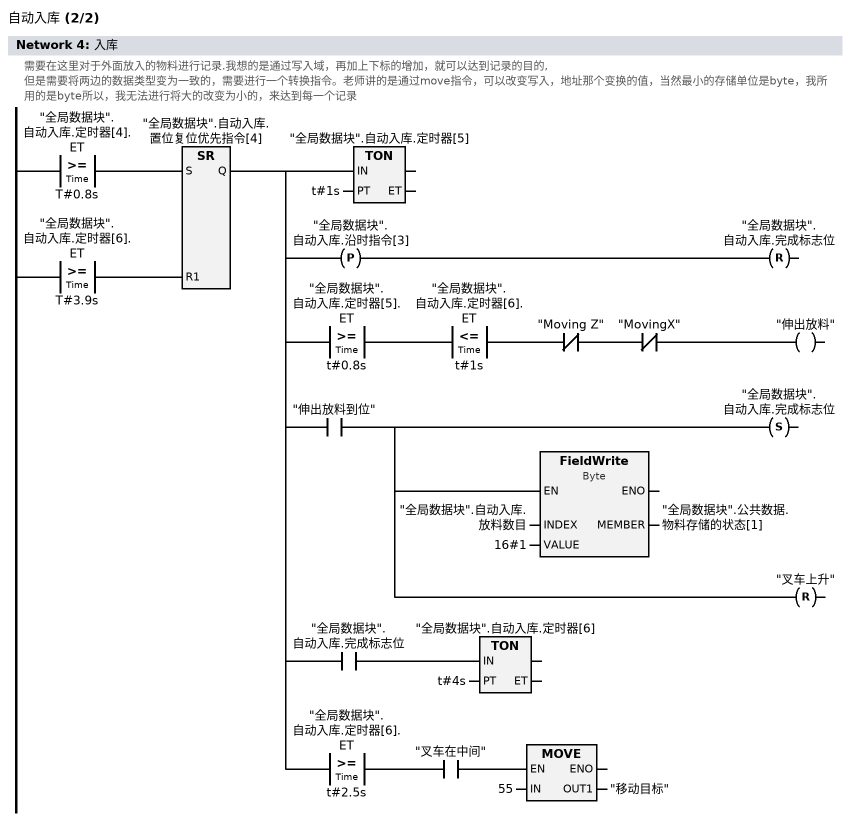
   // no SCL statement known for FieldWrite: written as a call
   IF "全局数据块".自动入库.定时器[4].ET >= T#0.8s THEN
       "全局数据块".自动入库.置位复位优先指令[4] := TRUE;   // SR flip-flop
   END_IF;
   IF "全局数据块".自动入库.定时器[6].ET >= T#3.9s THEN "全局数据块".自动入库.置位复位优先指令[4] := FALSE; END_IF;
   "全局数据块".自动入库.定时器[5].TON(IN := "全局数据块".自动入库.置位复位优先指令[4], PT := t#1s);
   #_w1 := "全局数据块".自动入库.置位复位优先指令[4] AND NOT "全局数据块".自动入库.沿时指令[3];   // rising edge
   "全局数据块".自动入库.沿时指令[3] := "全局数据块".自动入库.置位复位优先指令[4];
   IF #_w1 THEN "全局数据块".自动入库.完成标志位 := FALSE; END_IF;
   "伸出放料" := "全局数据块".自动入库.置位复位优先指令[4] AND ("全局数据块".自动入库.定时器[5].ET >= t#0.8s) AND ("全局数据块".自动入库.定时器[6].ET <= t#1s) AND NOT "Moving Z" AND NOT "MovingX";
   IF "全局数据块".自动入库.置位复位优先指令[4] AND "伸出放料到位" THEN "全局数据块".自动入库.完成标志位 := TRUE; END_IF;
   #_w2 := "全局数据块".自动入库.置位复位优先指令[4];
   #_w3 := "全局数据块".自动入库.置位复位优先指令[4] AND "伸出放料到位";
   IF #_w3 THEN
       FieldWrite(index := "全局数据块".自动入库.放料数目, value := 16#1, member => "全局数据块".公共数据.物料存储的状态[1]);
       "叉车上升" := FALSE;
   END_IF;
   "全局数据块".自动入库.定时器[6].TON(IN := #_w2 AND "全局数据块".自动入库.完成标志位, PT := t#4s);
   IF #_w2 AND ("全局数据块".自动入库.定时器[6].ET >= t#2.5s) AND "叉车在中间" THEN "移动目标" := 55; END_IF;
END_REGION
END_FUNCTION

// folder: 自动出库

FUNCTION "块_自动出库" : Void   // FC5, LAD
{ S7_Optimized_Access := 'TRUE' }
VERSION : 0.1
   VAR_TEMP   // added for the SCL form of the ladder/FBD networks
      _w1 : Bool;
      _w2 : Bool;
      _w3 : Bool;
      _w4 : Bool;
      _w5 : Bool;
      _w6 : Bool;
   END_VAR
BEGIN

REGION Network 1
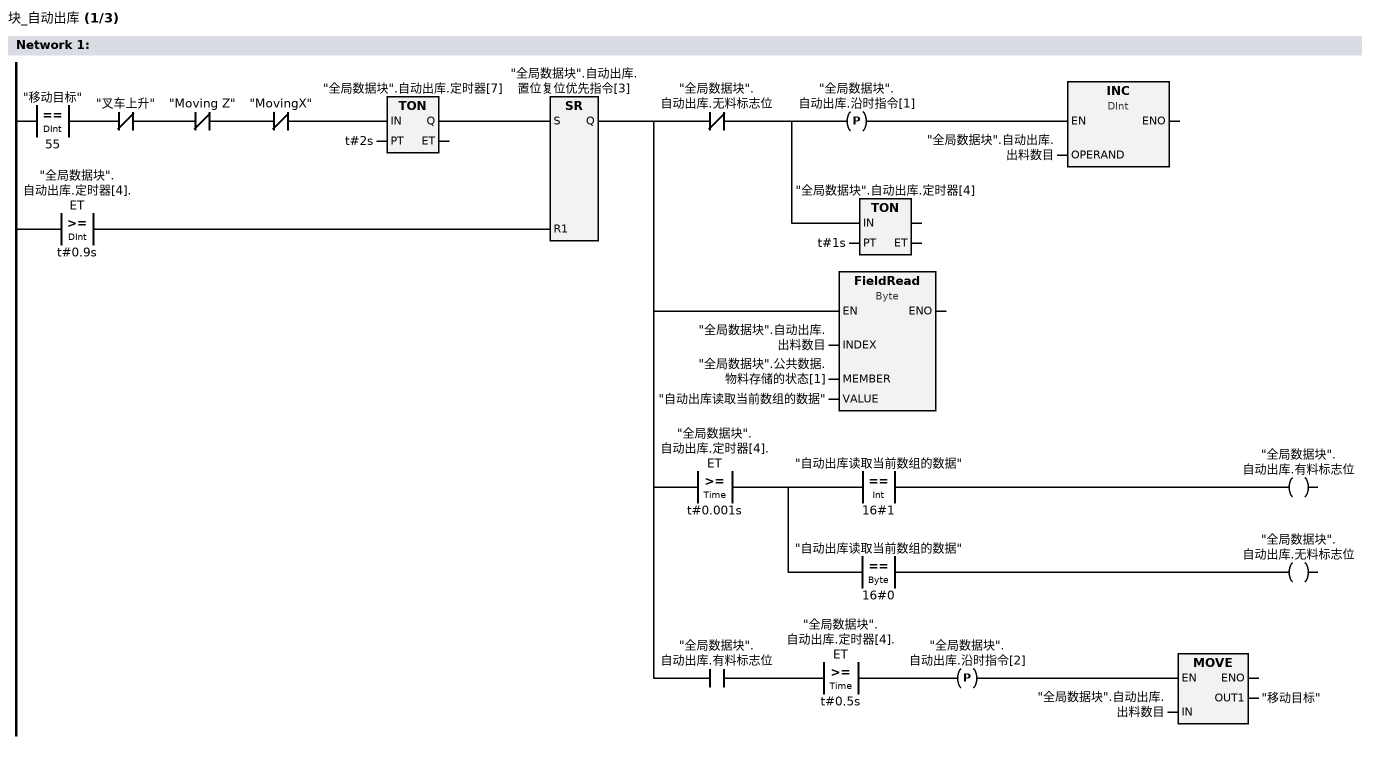
   // no SCL statement known for FieldRead: written as a call
   "全局数据块".自动出库.定时器[7].TON(IN := ("移动目标" = 55) AND NOT "叉车上升" AND NOT "Moving Z" AND NOT "MovingX", PT := t#2s);
   IF "全局数据块".自动出库.定时器[7].Q THEN
       "全局数据块".自动出库.置位复位优先指令[3] := TRUE;   // SR flip-flop
   END_IF;
   IF "全局数据块".自动出库.定时器[4].ET >= t#0.9s THEN "全局数据块".自动出库.置位复位优先指令[3] := FALSE; END_IF;
   #_w1 := "全局数据块".自动出库.置位复位优先指令[3] AND NOT "全局数据块".自动出库.无料标志位;
   #_w2 := #_w1 AND NOT "全局数据块".自动出库.沿时指令[1];   // rising edge
   "全局数据块".自动出库.沿时指令[1] := #_w1;
   IF #_w2 THEN "全局数据块".自动出库.出料数目 := "全局数据块".自动出库.出料数目 + 1; END_IF;
   "全局数据块".自动出库.定时器[4].TON(IN := #_w1, PT := t#1s);
   #_w3 := "全局数据块".自动出库.置位复位优先指令[3];
   IF #_w3 THEN
       FieldRead(index := "全局数据块".自动出库.出料数目, member := "全局数据块".公共数据.物料存储的状态[1], value := "自动出库读取当前数组的数据");
   END_IF;
   #_w4 := #_w3 AND ("全局数据块".自动出库.定时器[4].ET >= t#0.001s);
   "全局数据块".自动出库.有料标志位 := #_w4 AND ("自动出库读取当前数组的数据" = 16#1);
   "全局数据块".自动出库.无料标志位 := #_w4 AND ("自动出库读取当前数组的数据" = 16#0);
   #_w5 := #_w3 AND "全局数据块".自动出库.有料标志位 AND ("全局数据块".自动出库.定时器[4].ET >= t#0.5s);
   #_w6 := #_w5 AND NOT "全局数据块".自动出库.沿时指令[2];   // rising edge
   "全局数据块".自动出库.沿时指令[2] := #_w5;
   IF #_w6 THEN "移动目标" := "全局数据块".自动出库.出料数目; END_IF;
END_REGION

REGION Network 2: 入库
   // 需要在这里对于外面放入的物料进行记录.我想的是通过写入域，再加上下标的增加，就可以达到记录的目的,但是需要将两边的数据类型变为一致的，需要进行一个转换指令。老师讲的是通过move指令，可以改变写入，地址那个变换的值，当然最小的存储单位是byte，我所用的是byte所以，我无法进行将大的改变为小的，来达到每一个记录
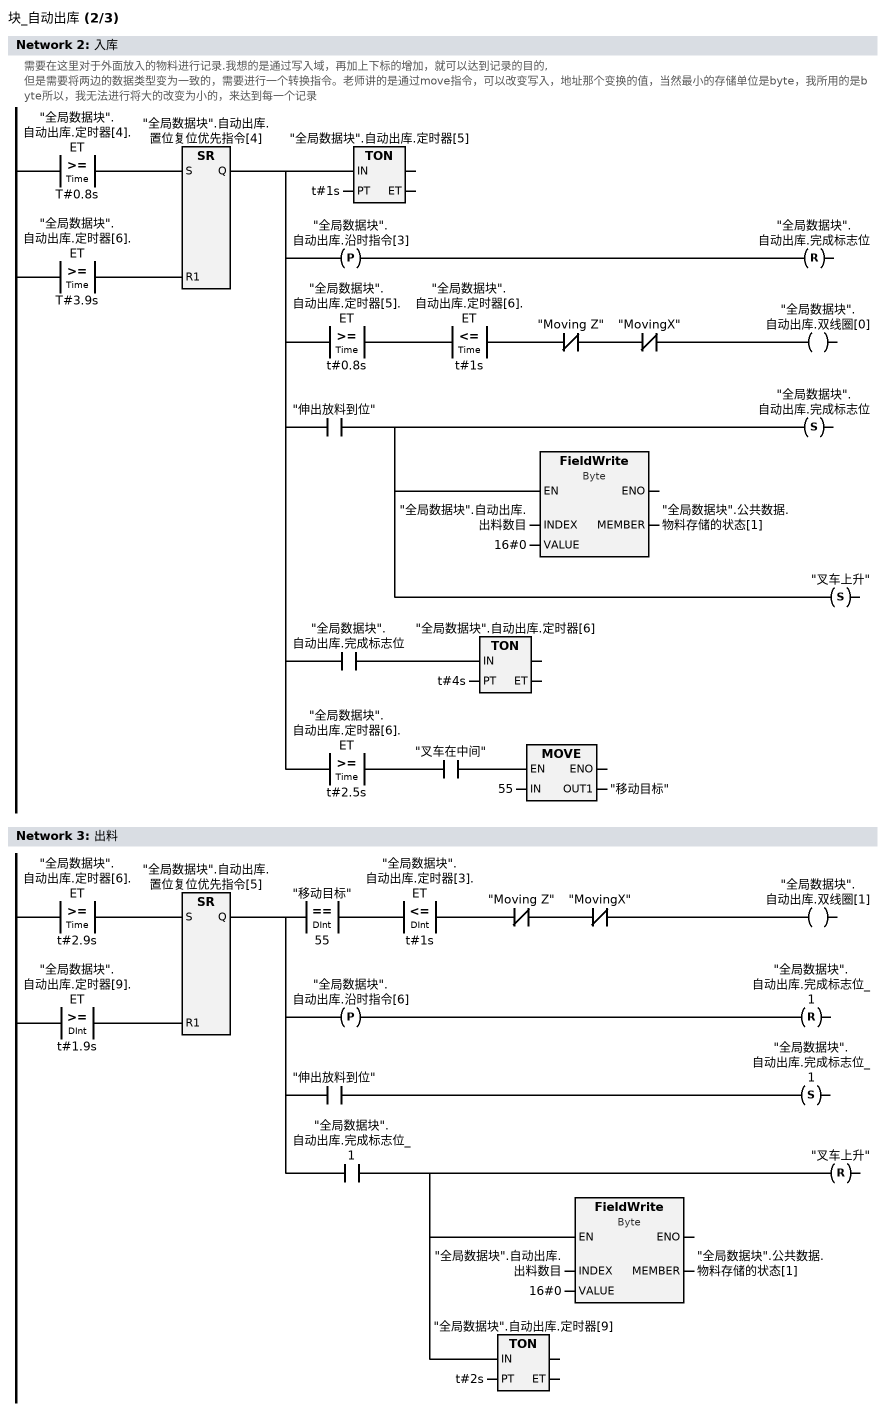
   // no SCL statement known for FieldWrite: written as a call
   IF "全局数据块".自动出库.定时器[4].ET >= T#0.8s THEN
       "全局数据块".自动出库.置位复位优先指令[4] := TRUE;   // SR flip-flop
   END_IF;
   IF "全局数据块".自动出库.定时器[6].ET >= T#3.9s THEN "全局数据块".自动出库.置位复位优先指令[4] := FALSE; END_IF;
   "全局数据块".自动出库.定时器[5].TON(IN := "全局数据块".自动出库.置位复位优先指令[4], PT := t#1s);
   #_w1 := "全局数据块".自动出库.置位复位优先指令[4] AND NOT "全局数据块".自动出库.沿时指令[3];   // rising edge
   "全局数据块".自动出库.沿时指令[3] := "全局数据块".自动出库.置位复位优先指令[4];
   IF #_w1 THEN "全局数据块".自动出库.完成标志位 := FALSE; END_IF;
   "全局数据块".自动出库.双线圈[0] := "全局数据块".自动出库.置位复位优先指令[4] AND ("全局数据块".自动出库.定时器[5].ET >= t#0.8s) AND ("全局数据块".自动出库.定时器[6].ET <= t#1s) AND NOT "Moving Z" AND NOT "MovingX";
   IF "全局数据块".自动出库.置位复位优先指令[4] AND "伸出放料到位" THEN "全局数据块".自动出库.完成标志位 := TRUE; END_IF;
   #_w2 := "全局数据块".自动出库.置位复位优先指令[4];
   #_w3 := "全局数据块".自动出库.置位复位优先指令[4] AND "伸出放料到位";
   IF #_w3 THEN
       FieldWrite(index := "全局数据块".自动出库.出料数目, value := 16#0, member => "全局数据块".公共数据.物料存储的状态[1]);
       "叉车上升" := TRUE;
   END_IF;
   "全局数据块".自动出库.定时器[6].TON(IN := #_w2 AND "全局数据块".自动出库.完成标志位, PT := t#4s);
   IF #_w2 AND ("全局数据块".自动出库.定时器[6].ET >= t#2.5s) AND "叉车在中间" THEN "移动目标" := 55; END_IF;
END_REGION

REGION Network 3: 出料
   // no SCL statement known for FieldWrite: written as a call
   IF "全局数据块".自动出库.定时器[6].ET >= t#2.9s THEN
       "全局数据块".自动出库.置位复位优先指令[5] := TRUE;   // SR flip-flop
   END_IF;
   IF "全局数据块".自动出库.定时器[9].ET >= t#1.9s THEN "全局数据块".自动出库.置位复位优先指令[5] := FALSE; END_IF;
   "全局数据块".自动出库.双线圈[1] := "全局数据块".自动出库.置位复位优先指令[5] AND ("移动目标" = 55) AND ("全局数据块".自动出库.定时器[3].ET <= t#1s) AND NOT "Moving Z" AND NOT "MovingX";
   #_w1 := "全局数据块".自动出库.置位复位优先指令[5] AND NOT "全局数据块".自动出库.沿时指令[6];   // rising edge
   "全局数据块".自动出库.沿时指令[6] := "全局数据块".自动出库.置位复位优先指令[5];
   IF #_w1 THEN "全局数据块".自动出库.完成标志位_1 := FALSE; END_IF;
   IF "全局数据块".自动出库.置位复位优先指令[5] AND "伸出放料到位" THEN "全局数据块".自动出库.完成标志位_1 := TRUE; END_IF;
   #_w2 := "全局数据块".自动出库.置位复位优先指令[5] AND "全局数据块".自动出库.完成标志位_1;
   IF #_w2 THEN
       "叉车上升" := FALSE;
       FieldWrite(index := "全局数据块".自动出库.出料数目, value := 16#0, member => "全局数据块".公共数据.物料存储的状态[1]);
   END_IF;
   "全局数据块".自动出库.定时器[9].TON(IN := #_w2, PT := t#2s);
END_REGION

REGION Network 4
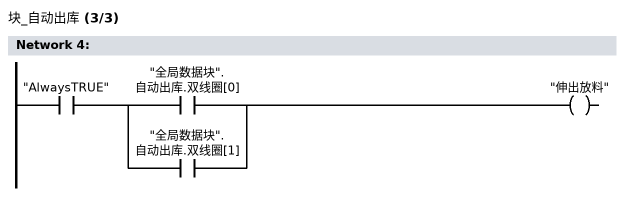
   RUNG wire#powerrail
      Contact( "AlwaysTRUE" )
      wire#w1
      Contact( "全局数据块".自动出库.双线圈[0] )
      wire#w2
      Coil( "伸出放料" )
   END_RUNG
   RUNG wire#w1
      Contact( "全局数据块".自动出库.双线圈[1] )
   END_RUNG wire#w2
   // the same network as SCL:
   "伸出放料" := "AlwaysTRUE" AND ("全局数据块".自动出库.双线圈[0] OR "全局数据块".自动出库.双线圈[1]);
END_REGION
END_FUNCTION

(* ===== HMI "HMI_RT_2" =====
system functions are stored by id; their names below are inferred from use
connection "HMI_连接_2": ETHERNET, S7_1200_OMS

HMI tags "默认变量表"
   "Tag_ScreenNumber" : UInt, internal
      on ChangeValue: ActivateScreenByNumber("动画列表", 0)
   "动画列表" : Int = PLC 动画列表 AT %MW100, 100 ms
      on ChangeValue: ActivateScreenByNumber("动画列表", 0)
   "入库手/自动开关" : Bool = PLC "入库手/自动开关" AT %M10.0, 1 s
   "自动运行指示灯" : Bool = PLC 自动运行指示灯 AT %M10.1, 1 s
   "手动运行指示灯" : Bool = PLC 手动运行指示灯 AT %M10.2, 1 s
   "全局数据块_公共数据_物料存储的状态{1}" : Byte = PLC 全局数据块.公共数据.物料存储的状态[1], 1 s
   "全局数据块_公共数据_物料存储的状态{2}" : Byte = PLC 全局数据块.公共数据.物料存储的状态[2], 1 s
   "全局数据块_公共数据_物料存储的状态{3}" : Byte = PLC 全局数据块.公共数据.物料存储的状态[3], 1 s
   "全局数据块_公共数据_物料存储的状态{4}" : Byte = PLC 全局数据块.公共数据.物料存储的状态[4], 1 s
   "全局数据块_公共数据_物料存储的状态{5}" : Byte = PLC 全局数据块.公共数据.物料存储的状态[5], 1 s
   "全局数据块_公共数据_物料存储的状态{6}" : Byte = PLC 全局数据块.公共数据.物料存储的状态[6], 1 s
   "全局数据块_公共数据_物料存储的状态{7}" : Byte = PLC 全局数据块.公共数据.物料存储的状态[7], 1 s
   "全局数据块_公共数据_物料存储的状态{8}" : Byte = PLC 全局数据块.公共数据.物料存储的状态[8], 1 s
   "全局数据块_公共数据_物料存储的状态{9}" : Byte = PLC 全局数据块.公共数据.物料存储的状态[9], 1 s
   "全局数据块_公共数据_物料存储的状态{10}" : Byte = PLC 全局数据块.公共数据.物料存储的状态[10], 1 s
   "全局数据块_公共数据_物料存储的状态{11}" : Byte = PLC 全局数据块.公共数据.物料存储的状态[11], 1 s
   "全局数据块_公共数据_物料存储的状态{12}" : Byte = PLC 全局数据块.公共数据.物料存储的状态[12], 1 s
   "全局数据块_公共数据_物料存储的状态{13}" : Byte = PLC 全局数据块.公共数据.物料存储的状态[13], 1 s
   "全局数据块_公共数据_物料存储的状态{14}" : Byte = PLC 全局数据块.公共数据.物料存储的状态[14], 1 s
   "全局数据块_公共数据_物料存储的状态{15}" : Byte = PLC 全局数据块.公共数据.物料存储的状态[15], 1 s
   "全局数据块_公共数据_物料存储的状态{16}" : Byte = PLC 全局数据块.公共数据.物料存储的状态[16], 1 s
   "全局数据块_公共数据_物料存储的状态{17}" : Byte = PLC 全局数据块.公共数据.物料存储的状态[17], 1 s
   "全局数据块_公共数据_物料存储的状态{18}" : Byte = PLC 全局数据块.公共数据.物料存储的状态[18], 1 s
   "全局数据块_公共数据_物料存储的状态{19}" : Byte = PLC 全局数据块.公共数据.物料存储的状态[19], 1 s
   "全局数据块_公共数据_物料存储的状态{20}" : Byte = PLC 全局数据块.公共数据.物料存储的状态[20], 1 s
   "全局数据块_公共数据_物料存储的状态{21}" : Byte = PLC 全局数据块.公共数据.物料存储的状态[21], 1 s
   "全局数据块_公共数据_物料存储的状态{22}" : Byte = PLC 全局数据块.公共数据.物料存储的状态[22], 1 s
   "全局数据块_公共数据_物料存储的状态{23}" : Byte = PLC 全局数据块.公共数据.物料存储的状态[23], 1 s
   "全局数据块_公共数据_物料存储的状态{24}" : Byte = PLC 全局数据块.公共数据.物料存储的状态[24], 1 s
   "全局数据块_公共数据_物料存储的状态{25}" : Byte = PLC 全局数据块.公共数据.物料存储的状态[25], 1 s
   "全局数据块_公共数据_物料存储的状态{26}" : Byte = PLC 全局数据块.公共数据.物料存储的状态[26], 1 s
   "全局数据块_公共数据_物料存储的状态{27}" : Byte = PLC 全局数据块.公共数据.物料存储的状态[27], 1 s
   "全局数据块_公共数据_物料存储的状态{28}" : Byte = PLC 全局数据块.公共数据.物料存储的状态[28], 1 s
   "全局数据块_公共数据_物料存储的状态{29}" : Byte = PLC 全局数据块.公共数据.物料存储的状态[29], 1 s
   "全局数据块_公共数据_物料存储的状态{30}" : Byte = PLC 全局数据块.公共数据.物料存储的状态[30], 1 s
   "全局数据块_公共数据_物料存储的状态{31}" : Byte = PLC 全局数据块.公共数据.物料存储的状态[31], 1 s
   "全局数据块_公共数据_物料存储的状态{32}" : Byte = PLC 全局数据块.公共数据.物料存储的状态[32], 1 s
   "全局数据块_公共数据_物料存储的状态{33}" : Byte = PLC 全局数据块.公共数据.物料存储的状态[33], 1 s
   "全局数据块_公共数据_物料存储的状态{34}" : Byte = PLC 全局数据块.公共数据.物料存储的状态[34], 1 s
   "全局数据块_公共数据_物料存储的状态{35}" : Byte = PLC 全局数据块.公共数据.物料存储的状态[35], 1 s
   "全局数据块_公共数据_物料存储的状态{36}" : Byte = PLC 全局数据块.公共数据.物料存储的状态[36], 1 s
   "全局数据块_公共数据_物料存储的状态{37}" : Byte = PLC 全局数据块.公共数据.物料存储的状态[37], 1 s
   "全局数据块_公共数据_物料存储的状态{38}" : Byte = PLC 全局数据块.公共数据.物料存储的状态[38], 1 s
   "全局数据块_公共数据_物料存储的状态{39}" : Byte = PLC 全局数据块.公共数据.物料存储的状态[39], 1 s
   "全局数据块_公共数据_物料存储的状态{40}" : Byte = PLC 全局数据块.公共数据.物料存储的状态[40], 1 s
   "全局数据块_公共数据_物料存储的状态{41}" : Byte = PLC 全局数据块.公共数据.物料存储的状态[41], 1 s
   "全局数据块_公共数据_物料存储的状态{42}" : Byte = PLC 全局数据块.公共数据.物料存储的状态[42], 1 s
   "全局数据块_公共数据_物料存储的状态{43}" : Byte = PLC 全局数据块.公共数据.物料存储的状态[43], 1 s
   "全局数据块_公共数据_物料存储的状态{44}" : Byte = PLC 全局数据块.公共数据.物料存储的状态[44], 1 s
   "全局数据块_公共数据_物料存储的状态{45}" : Byte = PLC 全局数据块.公共数据.物料存储的状态[45], 1 s
   "全局数据块_公共数据_物料存储的状态{46}" : Byte = PLC 全局数据块.公共数据.物料存储的状态[46], 1 s
   "全局数据块_公共数据_物料存储的状态{47}" : Byte = PLC 全局数据块.公共数据.物料存储的状态[47], 1 s
   "全局数据块_公共数据_物料存储的状态{48}" : Byte = PLC 全局数据块.公共数据.物料存储的状态[48], 1 s
   "全局数据块_公共数据_物料存储的状态{49}" : Byte = PLC 全局数据块.公共数据.物料存储的状态[49], 1 s
   "全局数据块_公共数据_物料存储的状态{50}" : Byte = PLC 全局数据块.公共数据.物料存储的状态[50], 1 s
   "全局数据块_公共数据_物料存储的状态{51}" : Byte = PLC 全局数据块.公共数据.物料存储的状态[51], 1 s
   "全局数据块_公共数据_物料存储的状态{52}" : Byte = PLC 全局数据块.公共数据.物料存储的状态[52], 1 s
   "全局数据块_公共数据_物料存储的状态{53}" : Byte = PLC 全局数据块.公共数据.物料存储的状态[53], 1 s
   "全局数据块_公共数据_物料存储的状态{54}" : Byte = PLC 全局数据块.公共数据.物料存储的状态[54], 1 s
   "一段电机" : Bool = PLC 一段电机 AT %Q2.0, 1 s
   "二段电机" : Bool = PLC 二段电机 AT %Q2.1, 1 s
   "伸出取料" : Bool = PLC 伸出取料 AT %Q2.2, 1 s
   "伸出放料" : Bool = PLC 伸出放料 AT %Q2.5, 1 s
   "叉车上升" : Bool = PLC 叉车上升 AT %Q2.3, 1 s
   "发料" : Bool = PLC 发料 AT %Q2.4, 1 s
   "MovingX" : Bool = PLC MovingX AT %I2.5, 1 s
   "Moving Z" : Bool = PLC "Moving Z" AT %I2.6, 1 s
   "全局数据块_自动入库_放料数目" : DInt = PLC 全局数据块.自动入库.放料数目, 1 s
   "全局数据块_手动入库_设置取料第几行" : DInt = PLC 全局数据块.手动入库.设置取料第几行, 1 s
   "全局数据块_手动入库_设置取料第几列" : DInt = PLC 全局数据块.手动入库.设置取料第几列, 1 s
   "全局数据块_手动入库_取料位置" : DInt = PLC 全局数据块.手动入库.取料位置, 1 s
   "全局数据块_手动入库_空位启动标志位" : Bool = PLC 全局数据块.手动入库.空位启动标志位, 1 s
   "全局数据块_手动入库_手动入库开关" : Bool = PLC 全局数据块.手动入库.手动入库开关, 1 s
   "全局数据块_动画切换_主页" : Bool = PLC 全局数据块.动画切换.主页, 1 s
   "全局数据块_动画切换_入库" : Bool = PLC 全局数据块.动画切换.入库, 1 s
   "全局数据块_动画切换_出库" : Bool = PLC 全局数据块.动画切换.出库, 1 s
   "全局数据块_动画切换_io" : Bool = PLC 全局数据块.动画切换.io, 1 s
   "全局数据块_动画切换_系统设置" : Bool = PLC 全局数据块.动画切换.系统设置, 1 s
   "全局数据块_手动出库_手动出库开关" : Bool = PLC 全局数据块.手动出库.手动出库开关, 1 s
   "全局数据块_手动出库_取料位置" : DInt = PLC 全局数据块.手动出库.取料位置, 1 s
   "全局数据块_手动出库_设置取料第几行" : DInt = PLC 全局数据块.手动出库.设置取料第几行, 1 s
   "全局数据块_手动出库_设置取料第几列" : DInt = PLC 全局数据块.手动出库.设置取料第几列, 1 s
   "入库指示灯" : Bool = PLC 入库指示灯 AT %M10.4, 1 s
   "出库指示灯" : Bool = PLC 出库指示灯 AT %M10.5, 1 s
   "自动/手动出库开关" : Bool = PLC "自动/手动出库开关" AT %M10.6, 1 s
   "自动出库指示灯" : Bool = PLC 自动出库指示灯 AT %M11.0, 1 s
   "手动出库指示灯" : Bool = PLC 手动出库指示灯 AT %M10.7, 1 s
   "启动入库" : Bool = PLC 启动入库 AT %M100.0, 1 s
   "启动出库" : Bool = PLC 启动出库 AT %M100.1, 1 s
   "出库/入库切换开关" : Bool = PLC "出库/入库切换开关" AT %M10.3, 1 s
   "三段电机" : Bool = PLC 三段电机 AT %Q3.0, 1 s
   "四段电机" : Bool = PLC 四段电机 AT %Q3.1, 1 s

screen "主页" 800x419, template "模板_1"
   on GenerateScreen: SetTag("Tag_ScreenNumber", 1)
   Button "按钮_1" at 29,314 size 96x32; TextOff '主页'
      on Press: SetBit("全局数据块_动画切换_主页")
      on Release: ResetBit("全局数据块_动画切换_主页")
   Button "按钮_2" at 142,314 size 96x32; TextOff '入库'
      on Release: ResetBit("全局数据块_动画切换_入库")
      on Press: SetBit("全局数据块_动画切换_入库")
   Button "按钮_3" at 252,314 size 96x32; TextOff '出库'
      on Press: SetBit("全局数据块_动画切换_出库")
      on Release: ResetBit("全局数据块_动画切换_出库")
   Button "按钮_4" at 481,314 size 96x32; TextOff '系统设置'
      on Press: SetBit("全局数据块_动画切换_系统设置")
      on Release: ResetBit("全局数据块_动画切换_系统设置")
   Button "按钮_5" at 369,314 size 96x32; TextOff 'io'
      on Release: ResetBit("全局数据块_动画切换_io")
      on Press: SetBit("全局数据块_动画切换_io")
   Button "按钮_6" at 596,314 size 96x32; TextOff '注销'
   Button "按钮_7" at 139,136 size 123x70; TextOff '入库模式'
      on Click: ActivateScreen("入库", 0)
   Button "按钮_8" at 462,136 size 123x70; TextOff '出库模式'
      on Click: ActivateScreen("出库", 0)
   Switch "开关_1" at 312,149 size 98x44; CaptionText 'Switch'; TextOff '入库'; TextOn '出库'
      ProcessValue <- "出库/入库切换开关"
   Circle "圆_1" at 180,71 size 48x48
      Appearance <- "入库指示灯"
   Circle "圆_2" at 493,77 size 48x48
      Appearance <- "出库指示灯"

Template "模板_1" 800x419
   Button "退出" at 720,360 size 78x58; TextOff '退出'; PictureOff "ExitRuntime_TP700_Comfort_TR"; PictureOn "ExitRuntime_TP700_Comfort_TR"
      on Release: StopRuntime(0)
   Button "Template_Button" at 640,360 size 78x58; TextOff 'Text'
   Button "Template_Button_1" at 560,360 size 78x58; TextOff 'Text'
   Button "Template_Button_2" at 480,360 size 78x58; TextOff 'Text'
   Button "Template_Button_3" at 400,360 size 78x58; TextOff 'Text'
   Button "Template_Button_4" at 321,360 size 78x58; TextOff 'Text'
   Button "Template_Button_5" at 241,360 size 78x58; TextOff 'Text'
   Button "Template_Button_6" at 161,360 size 78x58; TextOff 'Text'
   Button "Template_Button_7" at 81,360 size 78x58; TextOff 'Text'
   Button "起始画面" at 1,360 size 78x58; TextOff '起始画面'; PictureOff "NavigateHome_TP700_Comfort_TR"; PictureOn "NavigateHome_TP700_Comfort_TR"
      on Release: ActivateScreen("主页", 0)
   Button "按钮_1" at 29,314 size 96x32; TextOff '主页'
      on Press: SetBit("全局数据块_动画切换_主页")
      on Release: ResetBit("全局数据块_动画切换_主页")
   Button "按钮_2" at 142,314 size 96x32; TextOff '入库'
      on Release: ResetBit("全局数据块_动画切换_入库")
      on Press: SetBit("全局数据块_动画切换_入库")
   Button "按钮_3" at 252,314 size 96x32; TextOff '出库'
      on Press: SetBit("全局数据块_动画切换_出库")
      on Release: ResetBit("全局数据块_动画切换_出库")
   Button "按钮_4" at 481,314 size 96x32; TextOff '系统设置'
      on Press: SetBit("全局数据块_动画切换_系统设置")
      on Release: ResetBit("全局数据块_动画切换_系统设置")
   Button "按钮_5" at 369,314 size 96x32; TextOff 'io'
      on Release: ResetBit("全局数据块_动画切换_io")
      on Press: SetBit("全局数据块_动画切换_io")
   Button "按钮_6" at 596,314 size 96x32; TextOff '注销'

screen "出库" 800x419, template "模板_1"
   Button "按钮_7" at 139,136 size 123x70; TextOff '自动出库'
      on Click: ActivateScreen("自动出库", 0)
      on Change: ActivateScreen("自动出库", 0)
   Button "按钮_8" at 462,136 size 123x70; TextOff '手动出库'
      on Click: ActivateScreen("出库", 0)
      on Change: ActivateScreen("手动出库", 0)
   Switch "开关_1" at 312,149 size 98x44; TextOn '手动'; CaptionText 'Switch'; TextOff '自动'
      ProcessValue <- "自动/手动出库开关"
   Circle "圆_1" at 180,71 size 48x48
      Appearance <- "自动出库指示灯"
   Circle "圆_2" at 493,77 size 48x48
      Appearance <- "手动出库指示灯"

screen "入库" 800x419, template "模板_1"
   Button "按钮_1" at 484,142 size 148x90; TextOff '手动入库'
      on Click: ActivateScreen("手动入库", 0)
   Button "按钮_2" at 113,142 size 148x90; TextOff '自动入库'
      on Click: ActivateScreen("自动入库", 0)
   Switch "开关_1" at 298,158 size 148x61; CaptionText 'Switch'; TextOff '自动'; TextOn '手动'
      ProcessValue <- "入库手/自动开关"
   Circle "圆_1" at 534,83 size 48x48
      Appearance <- "手动运行指示灯"
   Circle "圆_2" at 160,83 size 48x48
      Appearance <- "自动运行指示灯"

screen "手动出库" 800x419, template "模板_1"
   Rectangle "矩形_1" at 25,36 size 29x21
      Appearance <- "全局数据块_公共数据_物料存储的状态{54}"
   Rectangle "矩形_2" at 65,36 size 29x21
      Appearance <- "全局数据块_公共数据_物料存储的状态{53}"
   Rectangle "矩形_3" at 105,36 size 29x21
      Appearance <- "全局数据块_公共数据_物料存储的状态{52}"
   Rectangle "矩形_4" at 145,36 size 29x21
      Appearance <- "全局数据块_公共数据_物料存储的状态{51}"
   Rectangle "矩形_5" at 185,36 size 29x21
      Appearance <- "全局数据块_公共数据_物料存储的状态{50}"
   Rectangle "矩形_6" at 225,36 size 29x21
      Appearance <- "全局数据块_公共数据_物料存储的状态{49}"
   Rectangle "矩形_7" at 265,36 size 29x21
      Appearance <- "全局数据块_公共数据_物料存储的状态{48}"
   Rectangle "矩形_8" at 305,36 size 29x21
      Appearance <- "全局数据块_公共数据_物料存储的状态{47}"
   Rectangle "矩形_9" at 345,36 size 29x21
      Appearance <- "全局数据块_公共数据_物料存储的状态{46}"
   Rectangle "矩形_10" at 25,76 size 29x21
      Appearance <- "全局数据块_公共数据_物料存储的状态{45}"
   Rectangle "矩形_11" at 65,76 size 29x21
      Appearance <- "全局数据块_公共数据_物料存储的状态{44}"
   Rectangle "矩形_12" at 105,76 size 29x21
      Appearance <- "全局数据块_公共数据_物料存储的状态{43}"
   Rectangle "矩形_13" at 145,76 size 29x21
      Appearance <- "全局数据块_公共数据_物料存储的状态{42}"
   Rectangle "矩形_14" at 185,76 size 29x21
      Appearance <- "全局数据块_公共数据_物料存储的状态{41}"
   Rectangle "矩形_15" at 225,76 size 29x21
      Appearance <- "全局数据块_公共数据_物料存储的状态{40}"
   Rectangle "矩形_16" at 265,76 size 29x21
      Appearance <- "全局数据块_公共数据_物料存储的状态{39}"
   Rectangle "矩形_17" at 305,76 size 29x21
      Appearance <- "全局数据块_公共数据_物料存储的状态{38}"
   Rectangle "矩形_18" at 345,76 size 29x21
      Appearance <- "全局数据块_公共数据_物料存储的状态{37}"
   Rectangle "矩形_19" at 24,111 size 29x21
      Appearance <- "全局数据块_公共数据_物料存储的状态{36}"
   Rectangle "矩形_20" at 64,111 size 29x21
      Appearance <- "全局数据块_公共数据_物料存储的状态{35}"
   Rectangle "矩形_21" at 104,111 size 29x21
      Appearance <- "全局数据块_公共数据_物料存储的状态{34}"
   Rectangle "矩形_22" at 144,111 size 29x21
      Appearance <- "全局数据块_公共数据_物料存储的状态{33}"
   Rectangle "矩形_23" at 184,111 size 29x21
      Appearance <- "全局数据块_公共数据_物料存储的状态{32}"
   Rectangle "矩形_24" at 224,111 size 29x21
      Appearance <- "全局数据块_公共数据_物料存储的状态{31}"
   Rectangle "矩形_25" at 264,111 size 29x21
      Appearance <- "全局数据块_公共数据_物料存储的状态{30}"
   Rectangle "矩形_26" at 304,111 size 29x21
      Appearance <- "全局数据块_公共数据_物料存储的状态{29}"
   Rectangle "矩形_27" at 344,111 size 29x21
      Appearance <- "全局数据块_公共数据_物料存储的状态{28}"
   Rectangle "矩形_28" at 25,151 size 29x21
      Appearance <- "全局数据块_公共数据_物料存储的状态{27}"
   Rectangle "矩形_29" at 65,151 size 29x21
      Appearance <- "全局数据块_公共数据_物料存储的状态{26}"
   Rectangle "矩形_30" at 105,151 size 29x21
      Appearance <- "全局数据块_公共数据_物料存储的状态{25}"
   Rectangle "矩形_31" at 145,151 size 29x21
      Appearance <- "全局数据块_公共数据_物料存储的状态{24}"
   Rectangle "矩形_32" at 185,151 size 29x21
      Appearance <- "全局数据块_公共数据_物料存储的状态{23}"
   Rectangle "矩形_33" at 225,151 size 29x21
      Appearance <- "全局数据块_公共数据_物料存储的状态{22}"
   Rectangle "矩形_34" at 265,151 size 29x21
      Appearance <- "全局数据块_公共数据_物料存储的状态{21}"
   Rectangle "矩形_35" at 305,151 size 29x21
      Appearance <- "全局数据块_公共数据_物料存储的状态{20}"
   Rectangle "矩形_36" at 345,151 size 29x21
      Appearance <- "全局数据块_公共数据_物料存储的状态{19}"
   Rectangle "矩形_37" at 26,191 size 29x21
      Appearance <- "全局数据块_公共数据_物料存储的状态{18}"
   Rectangle "矩形_38" at 66,191 size 29x21
      Appearance <- "全局数据块_公共数据_物料存储的状态{17}"
   Rectangle "矩形_39" at 106,191 size 29x21
      Appearance <- "全局数据块_公共数据_物料存储的状态{16}"
   Rectangle "矩形_40" at 146,191 size 29x21
      Appearance <- "全局数据块_公共数据_物料存储的状态{15}"
   Rectangle "矩形_41" at 186,191 size 29x21
      Appearance <- "全局数据块_公共数据_物料存储的状态{14}"
   Rectangle "矩形_42" at 226,191 size 29x21
      Appearance <- "全局数据块_公共数据_物料存储的状态{13}"
   Rectangle "矩形_43" at 266,191 size 29x21
      Appearance <- "全局数据块_公共数据_物料存储的状态{12}"
   Rectangle "矩形_44" at 306,191 size 29x21
      Appearance <- "全局数据块_公共数据_物料存储的状态{11}"
   Rectangle "矩形_45" at 346,191 size 29x21
      Appearance <- "全局数据块_公共数据_物料存储的状态{10}"
   Rectangle "矩形_46" at 27,231 size 29x21
      Appearance <- "全局数据块_公共数据_物料存储的状态{9}"
   Rectangle "矩形_47" at 67,231 size 29x21
      Appearance <- "全局数据块_公共数据_物料存储的状态{8}"
   Rectangle "矩形_48" at 107,231 size 29x21
      Appearance <- "全局数据块_公共数据_物料存储的状态{7}"
   Rectangle "矩形_49" at 147,231 size 29x21
      Appearance <- "全局数据块_公共数据_物料存储的状态{6}"
   Rectangle "矩形_50" at 187,231 size 29x21
      Appearance <- "全局数据块_公共数据_物料存储的状态{5}"
   Rectangle "矩形_51" at 227,231 size 29x21
      Appearance <- "全局数据块_公共数据_物料存储的状态{4}"
   Rectangle "矩形_52" at 267,231 size 29x21
      Appearance <- "全局数据块_公共数据_物料存储的状态{3}"
   Rectangle "矩形_53" at 307,231 size 29x21
      Appearance <- "全局数据块_公共数据_物料存储的状态{2}"
   Rectangle "矩形_54" at 347,231 size 29x21
      Appearance <- "全局数据块_公共数据_物料存储的状态{1}"
   TextField "文本域_3" at 354,16 size 14x20; Text '1'
   TextField "文本域_4" at 314,16 size 14x20; Text '2'
   TextField "文本域_5" at 274,16 size 14x20; Text '3'
   TextField "文本域_6" at 234,16 size 14x20; Text '4'
   TextField "文本域_7" at 194,16 size 14x20; Text '5'
   TextField "文本域_8" at 154,16 size 14x20; Text '6'
   TextField "文本域_9" at 114,16 size 14x20; Text '7'
   TextField "文本域_10" at 74,16 size 14x20; Text '8'
   TextField "文本域_11" at 34,16 size 14x20; Text '9'
   TextField "文本域_12" at 377,231 size 14x20; Text '1'
   TextField "文本域_13" at 354,16 size 14x20; Text '1'
   TextField "文本域_14" at 377,195 size 14x20; Text '2'
   TextField "文本域_15" at 377,149 size 14x20; Text '3'
   TextField "文本域_16" at 378,112 size 14x20; Text '4'
   TextField "文本域_17" at 377,76 size 14x20; Text '5'
   TextField "文本域_18" at 378,37 size 14x20; Text '6'
   TextField "文本域_2" at 377,263 size 56x20; Text '当前行'
   TextField "文本域_19" at 527,41 size 107x20; Text '放料位置设置'
   TextField "文本域_20" at 482,93 size 56x20; Text '放料第'
   TextField "文本域_21" at 482,149 size 56x20; Text '放料第'
   IOField "I/O 域_1" at 549,93 size 33x32; FormatPattern 99
      ProcessValue <- "全局数据块_手动出库_设置取料第几行"
   TextField "文本域_22" at 593,97 size 22x20; Text '行'
   IOField "I/O 域_2" at 549,149 size 33x32; FormatPattern 99
      ProcessValue <- "全局数据块_手动出库_设置取料第几列"
   TextField "文本域_23" at 588,149 size 22x20; Text '列'
   TextField "文本域_24" at 448,205 size 141x20; Text '设置移动当前位置'
   IOField "I/O 域_3" at 608,199 size 33x32; FormatPattern 99
      ProcessValue <- "全局数据块_手动出库_取料位置"
   Button "按钮_1" at 492,258 size 100x43; TextOff '放料开关'
      on Release: ResetBit("全局数据块_手动出库_手动出库开关")
      on Press: SetBit("全局数据块_手动出库_手动出库开关")
   TextField "文本域_1" at 0,0 size 56x20; Text '当前列'

screen "手动入库" 800x419, template "模板_1"
   Rectangle "矩形_1" at 25,36 size 29x21
      Appearance <- "全局数据块_公共数据_物料存储的状态{54}"
   Rectangle "矩形_2" at 65,36 size 29x21
      Appearance <- "全局数据块_公共数据_物料存储的状态{53}"
   Rectangle "矩形_3" at 105,36 size 29x21
      Appearance <- "全局数据块_公共数据_物料存储的状态{52}"
   Rectangle "矩形_4" at 145,36 size 29x21
      Appearance <- "全局数据块_公共数据_物料存储的状态{51}"
   Rectangle "矩形_5" at 185,36 size 29x21
      Appearance <- "全局数据块_公共数据_物料存储的状态{50}"
   Rectangle "矩形_6" at 225,36 size 29x21
      Appearance <- "全局数据块_公共数据_物料存储的状态{49}"
   Rectangle "矩形_7" at 265,36 size 29x21
      Appearance <- "全局数据块_公共数据_物料存储的状态{48}"
   Rectangle "矩形_8" at 305,36 size 29x21
      Appearance <- "全局数据块_公共数据_物料存储的状态{47}"
   Rectangle "矩形_9" at 345,36 size 29x21
      Appearance <- "全局数据块_公共数据_物料存储的状态{46}"
   Rectangle "矩形_10" at 25,76 size 29x21
      Appearance <- "全局数据块_公共数据_物料存储的状态{45}"
   Rectangle "矩形_11" at 65,76 size 29x21
      Appearance <- "全局数据块_公共数据_物料存储的状态{44}"
   Rectangle "矩形_12" at 105,76 size 29x21
      Appearance <- "全局数据块_公共数据_物料存储的状态{43}"
   Rectangle "矩形_13" at 145,76 size 29x21
      Appearance <- "全局数据块_公共数据_物料存储的状态{42}"
   Rectangle "矩形_14" at 185,76 size 29x21
      Appearance <- "全局数据块_公共数据_物料存储的状态{41}"
   Rectangle "矩形_15" at 225,76 size 29x21
      Appearance <- "全局数据块_公共数据_物料存储的状态{40}"
   Rectangle "矩形_16" at 265,76 size 29x21
      Appearance <- "全局数据块_公共数据_物料存储的状态{39}"
   Rectangle "矩形_17" at 305,76 size 29x21
      Appearance <- "全局数据块_公共数据_物料存储的状态{38}"
   Rectangle "矩形_18" at 345,76 size 29x21
      Appearance <- "全局数据块_公共数据_物料存储的状态{37}"
   Rectangle "矩形_19" at 24,111 size 29x21
      Appearance <- "全局数据块_公共数据_物料存储的状态{36}"
   Rectangle "矩形_20" at 64,111 size 29x21
      Appearance <- "全局数据块_公共数据_物料存储的状态{35}"
   Rectangle "矩形_21" at 104,111 size 29x21
      Appearance <- "全局数据块_公共数据_物料存储的状态{34}"
   Rectangle "矩形_22" at 144,111 size 29x21
      Appearance <- "全局数据块_公共数据_物料存储的状态{33}"
   Rectangle "矩形_23" at 184,111 size 29x21
      Appearance <- "全局数据块_公共数据_物料存储的状态{32}"
   Rectangle "矩形_24" at 224,111 size 29x21
      Appearance <- "全局数据块_公共数据_物料存储的状态{31}"
   Rectangle "矩形_25" at 264,111 size 29x21
      Appearance <- "全局数据块_公共数据_物料存储的状态{30}"
   Rectangle "矩形_26" at 304,111 size 29x21
      Appearance <- "全局数据块_公共数据_物料存储的状态{29}"
   Rectangle "矩形_27" at 344,111 size 29x21
      Appearance <- "全局数据块_公共数据_物料存储的状态{28}"
   Rectangle "矩形_28" at 25,151 size 29x21
      Appearance <- "全局数据块_公共数据_物料存储的状态{27}"
   Rectangle "矩形_29" at 65,151 size 29x21
      Appearance <- "全局数据块_公共数据_物料存储的状态{26}"
   Rectangle "矩形_30" at 105,151 size 29x21
      Appearance <- "全局数据块_公共数据_物料存储的状态{25}"
   Rectangle "矩形_31" at 145,151 size 29x21
      Appearance <- "全局数据块_公共数据_物料存储的状态{24}"
   Rectangle "矩形_32" at 185,151 size 29x21
      Appearance <- "全局数据块_公共数据_物料存储的状态{23}"
   Rectangle "矩形_33" at 225,151 size 29x21
      Appearance <- "全局数据块_公共数据_物料存储的状态{22}"
   Rectangle "矩形_34" at 265,151 size 29x21
      Appearance <- "全局数据块_公共数据_物料存储的状态{21}"
   Rectangle "矩形_35" at 305,151 size 29x21
      Appearance <- "全局数据块_公共数据_物料存储的状态{20}"
   Rectangle "矩形_36" at 345,151 size 29x21
      Appearance <- "全局数据块_公共数据_物料存储的状态{19}"
   Rectangle "矩形_37" at 26,191 size 29x21
      Appearance <- "全局数据块_公共数据_物料存储的状态{18}"
   Rectangle "矩形_38" at 66,191 size 29x21
      Appearance <- "全局数据块_公共数据_物料存储的状态{17}"
   Rectangle "矩形_39" at 106,191 size 29x21
      Appearance <- "全局数据块_公共数据_物料存储的状态{16}"
   Rectangle "矩形_40" at 146,191 size 29x21
      Appearance <- "全局数据块_公共数据_物料存储的状态{15}"
   Rectangle "矩形_41" at 186,191 size 29x21
      Appearance <- "全局数据块_公共数据_物料存储的状态{14}"
   Rectangle "矩形_42" at 226,191 size 29x21
      Appearance <- "全局数据块_公共数据_物料存储的状态{13}"
   Rectangle "矩形_43" at 266,191 size 29x21
      Appearance <- "全局数据块_公共数据_物料存储的状态{12}"
   Rectangle "矩形_44" at 306,191 size 29x21
      Appearance <- "全局数据块_公共数据_物料存储的状态{11}"
   Rectangle "矩形_45" at 346,191 size 29x21
      Appearance <- "全局数据块_公共数据_物料存储的状态{10}"
   Rectangle "矩形_46" at 27,231 size 29x21
      Appearance <- "全局数据块_公共数据_物料存储的状态{9}"
   Rectangle "矩形_47" at 67,231 size 29x21
      Appearance <- "全局数据块_公共数据_物料存储的状态{8}"
   Rectangle "矩形_48" at 107,231 size 29x21
      Appearance <- "全局数据块_公共数据_物料存储的状态{7}"
   Rectangle "矩形_49" at 147,231 size 29x21
      Appearance <- "全局数据块_公共数据_物料存储的状态{6}"
   Rectangle "矩形_50" at 187,231 size 29x21
      Appearance <- "全局数据块_公共数据_物料存储的状态{5}"
   Rectangle "矩形_51" at 227,231 size 29x21
      Appearance <- "全局数据块_公共数据_物料存储的状态{4}"
   Rectangle "矩形_52" at 267,231 size 29x21
      Appearance <- "全局数据块_公共数据_物料存储的状态{3}"
   Rectangle "矩形_53" at 307,231 size 29x21
      Appearance <- "全局数据块_公共数据_物料存储的状态{2}"
   Rectangle "矩形_54" at 347,231 size 29x21
      Appearance <- "全局数据块_公共数据_物料存储的状态{1}"
   TextField "文本域_1" at 6,5 size 56x20; Text '当前列'
   TextField "文本域_3" at 354,16 size 14x20; Text '1'
   TextField "文本域_4" at 314,16 size 14x20; Text '2'
   TextField "文本域_5" at 274,16 size 14x20; Text '3'
   TextField "文本域_6" at 234,16 size 14x20; Text '4'
   TextField "文本域_7" at 194,16 size 14x20; Text '5'
   TextField "文本域_8" at 154,16 size 14x20; Text '6'
   TextField "文本域_9" at 114,16 size 14x20; Text '7'
   TextField "文本域_10" at 74,16 size 14x20; Text '8'
   TextField "文本域_11" at 34,16 size 14x20; Text '9'
   TextField "文本域_12" at 377,231 size 14x20; Text '1'
   TextField "文本域_13" at 354,16 size 14x20; Text '1'
   TextField "文本域_14" at 377,195 size 14x20; Text '2'
   TextField "文本域_15" at 377,149 size 14x20; Text '3'
   TextField "文本域_16" at 378,112 size 14x20; Text '4'
   TextField "文本域_17" at 377,76 size 14x20; Text '5'
   TextField "文本域_18" at 378,37 size 14x20; Text '6'
   TextField "文本域_2" at 377,263 size 56x20; Text '当前行'
   TextField "文本域_19" at 527,41 size 107x20; Text '放料位置设置'
   TextField "文本域_20" at 482,93 size 56x20; Text '放料第'
   TextField "文本域_21" at 482,149 size 56x20; Text '放料第'
   IOField "I/O 域_1" at 549,93 size 33x32; FormatPattern 99
      ProcessValue <- "全局数据块_手动入库_设置取料第几行"
   TextField "文本域_22" at 593,97 size 22x20; Text '行'
   IOField "I/O 域_2" at 549,149 size 33x32; FormatPattern 99
      ProcessValue <- "全局数据块_手动入库_设置取料第几列"
   TextField "文本域_23" at 588,149 size 22x20; Text '列'
   TextField "文本域_24" at 448,205 size 141x20; Text '设置移动当前位置'
   IOField "I/O 域_3" at 608,199 size 33x32; FormatPattern 99
      ProcessValue <- "全局数据块_手动入库_取料位置"
   Button "按钮_1" at 492,258 size 100x43; TextOff '放料开关'
      on Press: SetBit("全局数据块_手动入库_手动入库开关")
      on Release: ResetBit("全局数据块_手动入库_手动入库开关")

screen "自动出库" 800x419, template "模板_1"
   Rectangle "矩形_1" at 25,36 size 29x21
      Appearance <- "全局数据块_公共数据_物料存储的状态{54}"
   Rectangle "矩形_2" at 65,36 size 29x21
      Appearance <- "全局数据块_公共数据_物料存储的状态{53}"
   Rectangle "矩形_3" at 105,36 size 29x21
      Appearance <- "全局数据块_公共数据_物料存储的状态{52}"
   Rectangle "矩形_4" at 145,36 size 29x21
      Appearance <- "全局数据块_公共数据_物料存储的状态{51}"
   Rectangle "矩形_5" at 185,36 size 29x21
      Appearance <- "全局数据块_公共数据_物料存储的状态{50}"
   Rectangle "矩形_6" at 225,36 size 29x21
      Appearance <- "全局数据块_公共数据_物料存储的状态{49}"
   Rectangle "矩形_7" at 265,36 size 29x21
      Appearance <- "全局数据块_公共数据_物料存储的状态{48}"
   Rectangle "矩形_8" at 305,36 size 29x21
      Appearance <- "全局数据块_公共数据_物料存储的状态{47}"
   Rectangle "矩形_9" at 345,36 size 29x21
      Appearance <- "全局数据块_公共数据_物料存储的状态{46}"
   Rectangle "矩形_10" at 25,76 size 29x21
      Appearance <- "全局数据块_公共数据_物料存储的状态{45}"
   Rectangle "矩形_11" at 65,76 size 29x21
      Appearance <- "全局数据块_公共数据_物料存储的状态{44}"
   Rectangle "矩形_12" at 105,76 size 29x21
      Appearance <- "全局数据块_公共数据_物料存储的状态{43}"
   Rectangle "矩形_13" at 145,76 size 29x21
      Appearance <- "全局数据块_公共数据_物料存储的状态{42}"
   Rectangle "矩形_14" at 185,76 size 29x21
      Appearance <- "全局数据块_公共数据_物料存储的状态{41}"
   Rectangle "矩形_15" at 225,76 size 29x21
      Appearance <- "全局数据块_公共数据_物料存储的状态{40}"
   Rectangle "矩形_16" at 265,76 size 29x21
      Appearance <- "全局数据块_公共数据_物料存储的状态{39}"
   Rectangle "矩形_17" at 305,76 size 29x21
      Appearance <- "全局数据块_公共数据_物料存储的状态{38}"
   Rectangle "矩形_18" at 345,76 size 29x21
      Appearance <- "全局数据块_公共数据_物料存储的状态{37}"
   Rectangle "矩形_19" at 24,111 size 29x21
      Appearance <- "全局数据块_公共数据_物料存储的状态{36}"
   Rectangle "矩形_20" at 64,111 size 29x21
      Appearance <- "全局数据块_公共数据_物料存储的状态{35}"
   Rectangle "矩形_21" at 104,111 size 29x21
      Appearance <- "全局数据块_公共数据_物料存储的状态{34}"
   Rectangle "矩形_22" at 144,111 size 29x21
      Appearance <- "全局数据块_公共数据_物料存储的状态{33}"
   Rectangle "矩形_23" at 184,111 size 29x21
      Appearance <- "全局数据块_公共数据_物料存储的状态{32}"
   Rectangle "矩形_24" at 224,111 size 29x21
      Appearance <- "全局数据块_公共数据_物料存储的状态{31}"
   Rectangle "矩形_25" at 264,111 size 29x21
      Appearance <- "全局数据块_公共数据_物料存储的状态{30}"
   Rectangle "矩形_26" at 304,111 size 29x21
      Appearance <- "全局数据块_公共数据_物料存储的状态{29}"
   Rectangle "矩形_27" at 344,111 size 29x21
      Appearance <- "全局数据块_公共数据_物料存储的状态{28}"
   Rectangle "矩形_28" at 25,151 size 29x21
      Appearance <- "全局数据块_公共数据_物料存储的状态{27}"
   Rectangle "矩形_29" at 65,151 size 29x21
      Appearance <- "全局数据块_公共数据_物料存储的状态{26}"
   Rectangle "矩形_30" at 105,151 size 29x21
      Appearance <- "全局数据块_公共数据_物料存储的状态{25}"
   Rectangle "矩形_31" at 145,151 size 29x21
      Appearance <- "全局数据块_公共数据_物料存储的状态{24}"
   Rectangle "矩形_32" at 185,151 size 29x21
      Appearance <- "全局数据块_公共数据_物料存储的状态{23}"
   Rectangle "矩形_33" at 225,151 size 29x21
      Appearance <- "全局数据块_公共数据_物料存储的状态{22}"
   Rectangle "矩形_34" at 265,151 size 29x21
      Appearance <- "全局数据块_公共数据_物料存储的状态{21}"
   Rectangle "矩形_35" at 305,151 size 29x21
      Appearance <- "全局数据块_公共数据_物料存储的状态{20}"
   Rectangle "矩形_36" at 345,151 size 29x21
      Appearance <- "全局数据块_公共数据_物料存储的状态{19}"
   Rectangle "矩形_37" at 26,191 size 29x21
      Appearance <- "全局数据块_公共数据_物料存储的状态{18}"
   Rectangle "矩形_38" at 66,191 size 29x21
      Appearance <- "全局数据块_公共数据_物料存储的状态{17}"
   Rectangle "矩形_39" at 106,191 size 29x21
      Appearance <- "全局数据块_公共数据_物料存储的状态{16}"
   Rectangle "矩形_40" at 146,191 size 29x21
      Appearance <- "全局数据块_公共数据_物料存储的状态{15}"
   Rectangle "矩形_41" at 186,191 size 29x21
      Appearance <- "全局数据块_公共数据_物料存储的状态{14}"
   Rectangle "矩形_42" at 226,191 size 29x21
      Appearance <- "全局数据块_公共数据_物料存储的状态{13}"
   Rectangle "矩形_43" at 266,191 size 29x21
      Appearance <- "全局数据块_公共数据_物料存储的状态{12}"
   Rectangle "矩形_44" at 306,191 size 29x21
      Appearance <- "全局数据块_公共数据_物料存储的状态{11}"
   Rectangle "矩形_45" at 346,191 size 29x21
      Appearance <- "全局数据块_公共数据_物料存储的状态{10}"
   Rectangle "矩形_46" at 27,231 size 29x21
      Appearance <- "全局数据块_公共数据_物料存储的状态{9}"
   Rectangle "矩形_47" at 67,231 size 29x21
      Appearance <- "全局数据块_公共数据_物料存储的状态{8}"
   Rectangle "矩形_48" at 107,231 size 29x21
      Appearance <- "全局数据块_公共数据_物料存储的状态{7}"
   Rectangle "矩形_49" at 147,231 size 29x21
      Appearance <- "全局数据块_公共数据_物料存储的状态{6}"
   Rectangle "矩形_50" at 187,231 size 29x21
      Appearance <- "全局数据块_公共数据_物料存储的状态{5}"
   Rectangle "矩形_51" at 227,231 size 29x21
      Appearance <- "全局数据块_公共数据_物料存储的状态{4}"
   Rectangle "矩形_52" at 267,231 size 29x21
      Appearance <- "全局数据块_公共数据_物料存储的状态{3}"
   Rectangle "矩形_53" at 307,231 size 29x21
      Appearance <- "全局数据块_公共数据_物料存储的状态{2}"
   Rectangle "矩形_54" at 347,231 size 29x21
      Appearance <- "全局数据块_公共数据_物料存储的状态{1}"
   TextField "文本域_2" at 354,264 size 56x20; Text '当前行'
   TextField "文本域_3" at 354,16 size 14x20; Text '1'
   TextField "文本域_4" at 314,16 size 14x20; Text '2'
   TextField "文本域_5" at 274,16 size 14x20; Text '3'
   TextField "文本域_6" at 234,16 size 14x20; Text '4'
   TextField "文本域_7" at 194,16 size 14x20; Text '5'
   TextField "文本域_8" at 154,16 size 14x20; Text '6'
   TextField "文本域_9" at 114,16 size 14x20; Text '7'
   TextField "文本域_10" at 74,16 size 14x20; Text '8'
   TextField "文本域_11" at 34,16 size 14x20; Text '9'
   TextField "文本域_12" at 377,231 size 14x20; Text '1'
   TextField "文本域_13" at 354,16 size 14x20; Text '1'
   TextField "文本域_14" at 377,195 size 14x20; Text '2'
   TextField "文本域_15" at 377,149 size 14x20; Text '3'
   TextField "文本域_16" at 378,112 size 14x20; Text '4'
   TextField "文本域_17" at 377,76 size 14x20; Text '5'
   TextField "文本域_18" at 378,37 size 14x20; Text '6'
   TextField "文本域_19" at 481,5 size 73x20; Text '动作状态'
   Circle "圆_1" at 409,25 size 35x35
      Appearance <- "三段电机"
   Circle "圆_2" at 409,69 size 35x35
      Appearance <- "四段电机"
   Circle "圆_3" at 409,110 size 35x35
      Appearance <- "伸出取料"
   Circle "圆_4" at 409,146 size 35x35
      Appearance <- "伸出放料"
   Circle "圆_5" at 409,193 size 35x35
      Appearance <- "叉车上升"
   Circle "圆_6" at 409,229 size 35x35
      Appearance <- "发料"
   TextField "文本域_20" at 449,38 size 69x19; Text '三段电机'
   TextField "文本域_21" at 449,78 size 69x19; Text '四段电机'
   TextField "文本域_22" at 450,122 size 69x19; Text '伸出取料'
   TextField "文本域_23" at 450,162 size 69x19; Text '伸出放料'
   TextField "文本域_24" at 450,209 size 69x19; Text '叉车上升'
   TextField "文本域_25" at 467,240 size 37x19; Text '出料'
   TextField "文本域_28" at 422,271 size 125x23; Text '当前物料标签'
   TextField "文本域_29" at 520,71 size 14x20; Text 'Text'
   Circle "圆_7" at 62,259 size 35x35
      Appearance <- "MovingX"
   Circle "圆_8" at 216,259 size 35x35
      Appearance <- "Moving Z"
   TextField "文本域_26" at 124,264 size 61x20; Text 'MovingX'
   TextField "文本域_27" at 266,264 size 61x20; Text 'MovingZ'

screen "自动入库" 800x419, template "模板_1"
   Rectangle "矩形_1" at 25,36 size 29x21
      Appearance <- "全局数据块_公共数据_物料存储的状态{54}"
   Rectangle "矩形_2" at 65,36 size 29x21
      Appearance <- "全局数据块_公共数据_物料存储的状态{53}"
   Rectangle "矩形_3" at 105,36 size 29x21
      Appearance <- "全局数据块_公共数据_物料存储的状态{52}"
   Rectangle "矩形_4" at 145,36 size 29x21
      Appearance <- "全局数据块_公共数据_物料存储的状态{51}"
   Rectangle "矩形_5" at 185,36 size 29x21
      Appearance <- "全局数据块_公共数据_物料存储的状态{50}"
   Rectangle "矩形_6" at 225,36 size 29x21
      Appearance <- "全局数据块_公共数据_物料存储的状态{49}"
   Rectangle "矩形_7" at 265,36 size 29x21
      Appearance <- "全局数据块_公共数据_物料存储的状态{48}"
   Rectangle "矩形_8" at 305,36 size 29x21
      Appearance <- "全局数据块_公共数据_物料存储的状态{47}"
   Rectangle "矩形_9" at 345,36 size 29x21
      Appearance <- "全局数据块_公共数据_物料存储的状态{46}"
   Rectangle "矩形_10" at 25,76 size 29x21
      Appearance <- "全局数据块_公共数据_物料存储的状态{45}"
   Rectangle "矩形_11" at 65,76 size 29x21
      Appearance <- "全局数据块_公共数据_物料存储的状态{44}"
   Rectangle "矩形_12" at 105,76 size 29x21
      Appearance <- "全局数据块_公共数据_物料存储的状态{43}"
   Rectangle "矩形_13" at 145,76 size 29x21
      Appearance <- "全局数据块_公共数据_物料存储的状态{42}"
   Rectangle "矩形_14" at 185,76 size 29x21
      Appearance <- "全局数据块_公共数据_物料存储的状态{41}"
   Rectangle "矩形_15" at 225,76 size 29x21
      Appearance <- "全局数据块_公共数据_物料存储的状态{40}"
   Rectangle "矩形_16" at 265,76 size 29x21
      Appearance <- "全局数据块_公共数据_物料存储的状态{39}"
   Rectangle "矩形_17" at 305,76 size 29x21
      Appearance <- "全局数据块_公共数据_物料存储的状态{38}"
   Rectangle "矩形_18" at 345,76 size 29x21
      Appearance <- "全局数据块_公共数据_物料存储的状态{37}"
   Rectangle "矩形_19" at 24,111 size 29x21
      Appearance <- "全局数据块_公共数据_物料存储的状态{36}"
   Rectangle "矩形_20" at 64,111 size 29x21
      Appearance <- "全局数据块_公共数据_物料存储的状态{35}"
   Rectangle "矩形_21" at 104,111 size 29x21
      Appearance <- "全局数据块_公共数据_物料存储的状态{34}"
   Rectangle "矩形_22" at 144,111 size 29x21
      Appearance <- "全局数据块_公共数据_物料存储的状态{33}"
   Rectangle "矩形_23" at 184,111 size 29x21
      Appearance <- "全局数据块_公共数据_物料存储的状态{32}"
   Rectangle "矩形_24" at 224,111 size 29x21
      Appearance <- "全局数据块_公共数据_物料存储的状态{31}"
   Rectangle "矩形_25" at 264,111 size 29x21
      Appearance <- "全局数据块_公共数据_物料存储的状态{30}"
   Rectangle "矩形_26" at 304,111 size 29x21
      Appearance <- "全局数据块_公共数据_物料存储的状态{29}"
   Rectangle "矩形_27" at 344,111 size 29x21
      Appearance <- "全局数据块_公共数据_物料存储的状态{28}"
   Rectangle "矩形_28" at 25,151 size 29x21
      Appearance <- "全局数据块_公共数据_物料存储的状态{27}"
   Rectangle "矩形_29" at 65,151 size 29x21
      Appearance <- "全局数据块_公共数据_物料存储的状态{26}"
   Rectangle "矩形_30" at 105,151 size 29x21
      Appearance <- "全局数据块_公共数据_物料存储的状态{25}"
   Rectangle "矩形_31" at 145,151 size 29x21
      Appearance <- "全局数据块_公共数据_物料存储的状态{24}"
   Rectangle "矩形_32" at 185,151 size 29x21
      Appearance <- "全局数据块_公共数据_物料存储的状态{23}"
   Rectangle "矩形_33" at 225,151 size 29x21
      Appearance <- "全局数据块_公共数据_物料存储的状态{22}"
   Rectangle "矩形_34" at 265,151 size 29x21
      Appearance <- "全局数据块_公共数据_物料存储的状态{21}"
   Rectangle "矩形_35" at 305,151 size 29x21
      Appearance <- "全局数据块_公共数据_物料存储的状态{20}"
   Rectangle "矩形_36" at 345,151 size 29x21
      Appearance <- "全局数据块_公共数据_物料存储的状态{19}"
   Rectangle "矩形_37" at 26,191 size 29x21
      Appearance <- "全局数据块_公共数据_物料存储的状态{18}"
   Rectangle "矩形_38" at 66,191 size 29x21
      Appearance <- "全局数据块_公共数据_物料存储的状态{17}"
   Rectangle "矩形_39" at 106,191 size 29x21
      Appearance <- "全局数据块_公共数据_物料存储的状态{16}"
   Rectangle "矩形_40" at 146,191 size 29x21
      Appearance <- "全局数据块_公共数据_物料存储的状态{15}"
   Rectangle "矩形_41" at 186,191 size 29x21
      Appearance <- "全局数据块_公共数据_物料存储的状态{14}"
   Rectangle "矩形_42" at 226,191 size 29x21
      Appearance <- "全局数据块_公共数据_物料存储的状态{13}"
   Rectangle "矩形_43" at 266,191 size 29x21
      Appearance <- "全局数据块_公共数据_物料存储的状态{12}"
   Rectangle "矩形_44" at 306,191 size 29x21
      Appearance <- "全局数据块_公共数据_物料存储的状态{11}"
   Rectangle "矩形_45" at 346,191 size 29x21
      Appearance <- "全局数据块_公共数据_物料存储的状态{10}"
   Rectangle "矩形_46" at 27,231 size 29x21
      Appearance <- "全局数据块_公共数据_物料存储的状态{9}"
   Rectangle "矩形_47" at 67,231 size 29x21
      Appearance <- "全局数据块_公共数据_物料存储的状态{8}"
   Rectangle "矩形_48" at 107,231 size 29x21
      Appearance <- "全局数据块_公共数据_物料存储的状态{7}"
   Rectangle "矩形_49" at 147,231 size 29x21
      Appearance <- "全局数据块_公共数据_物料存储的状态{6}"
   Rectangle "矩形_50" at 187,231 size 29x21
      Appearance <- "全局数据块_公共数据_物料存储的状态{5}"
   Rectangle "矩形_51" at 227,231 size 29x21
      Appearance <- "全局数据块_公共数据_物料存储的状态{4}"
   Rectangle "矩形_52" at 267,231 size 29x21
      Appearance <- "全局数据块_公共数据_物料存储的状态{3}"
   Rectangle "矩形_53" at 307,231 size 29x21
      Appearance <- "全局数据块_公共数据_物料存储的状态{2}"
   Rectangle "矩形_54" at 347,231 size 29x21
      Appearance <- "全局数据块_公共数据_物料存储的状态{1}"
   TextField "文本域_1" at 6,5 size 56x20; Text '当前列'
   TextField "文本域_2" at 354,264 size 56x20; Text '当前行'
   TextField "文本域_3" at 354,16 size 14x20; Text '1'
   TextField "文本域_4" at 314,16 size 14x20; Text '2'
   TextField "文本域_5" at 274,16 size 14x20; Text '3'
   TextField "文本域_6" at 234,16 size 14x20; Text '4'
   TextField "文本域_7" at 194,16 size 14x20; Text '5'
   TextField "文本域_8" at 154,16 size 14x20; Text '6'
   TextField "文本域_9" at 114,16 size 14x20; Text '7'
   TextField "文本域_10" at 74,16 size 14x20; Text '8'
   TextField "文本域_11" at 34,16 size 14x20; Text '9'
   TextField "文本域_12" at 377,231 size 14x20; Text '1'
   TextField "文本域_13" at 354,16 size 14x20; Text '1'
   TextField "文本域_14" at 377,195 size 14x20; Text '2'
   TextField "文本域_15" at 377,149 size 14x20; Text '3'
   TextField "文本域_16" at 378,112 size 14x20; Text '4'
   TextField "文本域_17" at 377,76 size 14x20; Text '5'
   TextField "文本域_18" at 378,37 size 14x20; Text '6'
   TextField "文本域_19" at 481,5 size 73x20; Text '动作状态'
   Circle "圆_1" at 409,25 size 35x35
      Appearance <- "一段电机"
   Circle "圆_2" at 409,69 size 35x35
      Appearance <- "二段电机"
   Circle "圆_3" at 409,110 size 35x35
      Appearance <- "伸出取料"
   Circle "圆_4" at 409,146 size 35x35
      Appearance <- "伸出放料"
   Circle "圆_5" at 409,193 size 35x35
      Appearance <- "叉车上升"
   Circle "圆_6" at 409,229 size 35x35
      Appearance <- "发料"
   TextField "文本域_20" at 449,38 size 69x19; Text '一段电机'
   TextField "文本域_21" at 449,78 size 69x19; Text '二段电机'
   TextField "文本域_22" at 450,122 size 69x19; Text '伸出取料'
   TextField "文本域_23" at 450,162 size 69x19; Text '伸出放料'
   TextField "文本域_24" at 450,209 size 69x19; Text '叉车上升'
   TextField "文本域_25" at 467,240 size 37x19; Text '发料'
   Circle "圆_7" at 62,259 size 35x35
      Appearance <- "MovingX"
   Circle "圆_8" at 216,259 size 35x35
      Appearance <- "Moving Z"
   TextField "文本域_26" at 124,264 size 61x20; Text 'MovingX'
   TextField "文本域_27" at 266,264 size 61x20; Text 'MovingZ'
   TextField "文本域_28" at 422,271 size 125x23; Text '当前物料标签'
   IOField "I/O 域_1" at 570,271 size 34x32; FormatPattern 99
      ProcessValue <- "全局数据块_自动入库_放料数目"
   TextField "文本域_29" at 520,71 size 14x20; Text 'Text'
*)